IF ptrTc2_EtherCAT^.Input.Command.EcCoeSdoRead.Enable THEN
	FB_EcCoeSdoRead_0(
					sNetId		:= ptrTc2_EtherCAT^.Input.Parameter.EcCoeSdoRead.sNetId, 
					nSlaveAddr	:= ptrTc2_EtherCAT^.Input.Parameter.EcCoeSdoRead.nSlaveAddr, 
					nSubIndex	:= ptrTc2_EtherCAT^.Input.Parameter.EcCoeSdoRead.nSubIndex, 
					nIndex		:= ptrTc2_EtherCAT^.Input.Parameter.EcCoeSdoRead.nIndex , 
					pDstBuf		:= ptrTc2_EtherCAT^.Input.Parameter.EcCoeSdoRead.pDstBuf, 
					cbBufLen	:= ptrTc2_EtherCAT^.Input.Parameter.EcCoeSdoRead.cbBufLen, 
					bExecute	:= TRUE ,
					tTimeout	:= ptrTc2_EtherCAT^.Input.Parameter.EcCoeSdoRead.tTimeout, 
					bBusy		=> ptrTc2_EtherCAT^.Output.Status.EcCoeSdoRead.bBusy , 
					bError		=> ptrTc2_EtherCAT^.Output.Status.EcCoeSdoRead.bError, 
					nErrId		=> ptrTc2_EtherCAT^.Output.Error.ErrorID
					);
END_IF

IF NOT 	ptrTc2_EtherCAT^.Output.Status.EcCoeSdoRead.bBusy OR ptrTc2_EtherCAT^.Output.Status.EcCoeSdoRead.bError THEN
	ptrTc2_EtherCAT^.Input.Command.EcCoeSdoRead.Enable := FALSE ;
	FB_EcCoeSdoRead_0.bExecute := FALSE ;
	ptrTc2_EtherCAT^.Output.Status.EcCoeSdoRead.bError := FALSE ;
	FB_EcCoeSdoRead_0();
END_IF

(*IF ptrTc2_EtherCAT^.Input.Command.EcCoeSdoWrite.Enable THEN
	FB_EcCoESdoWrite_0(
						sNetId		:= ptrTc2_EtherCAT^.Input.Parameter.EcCoeSdoWrite.sNetId, 
						nSlaveAddr	:= ptrTc2_EtherCAT^.Input.Parameter.EcCoeSdoWrite.nSlaveAddr, 
						nSubIndex	:= ptrTc2_EtherCAT^.Input.Parameter.EcCoeSdoWrite.nSubIndex, 
						nIndex		:= ptrTc2_EtherCAT^.Input.Parameter.EcCoeSdoWrite.nIndex, 
						pSrcBuf		:= ptrTc2_EtherCAT^.Input.Parameter.EcCoeSdoWrite.pSrcBuf, 
						cbBufLen	:= ptrTc2_EtherCAT^.Input.Parameter.EcCoeSdoWrite.cbBufLen, 
						bExecute	:= TRUE, 
						tTimeout	:= ptrTc2_EtherCAT^.Input.Parameter.EcCoeSdoWrite.tTimeout, 
						bBusy		=> ptrTc2_EtherCAT^.Output.Status.EcCoeSdoWrite.bBusy, 
						bError		=> ptrTc2_EtherCAT^.Output.Status.EcCoeSdoWrite.bError, 
						nErrId		=> ptrTc2_EtherCAT^.Output.Error.ErrorID
					);			
END_IF

IF NOT 	ptrTc2_EtherCAT^.Output.Status.EcCoeSdoWrite.bBusy OR ptrTc2_EtherCAT^.Output.Status.EcCoeSdoWrite.bError THEN
	ptrTc2_EtherCAT^.Input.Command.EcCoeSdoWrite.Enable := FALSE ;
	FB_EcCoESdoWrite_0.bExecute := FALSE ;
	ptrTc2_EtherCAT^.Output.Status.EcCoeSdoWrite.bError := FALSE ;
	FB_EcCoESdoWrite_0();
END_IF	*)

IF ptrTc2_EtherCAT^.Input.Command.EcSoeRead.Enable THEN
	FB_EcSoERead_0(
					sNetId		:= ptrTc2_EtherCAT^.Input.Parameter.EcSoeRead.sNetId, 
					nSlaveAddr	:= ptrTc2_EtherCAT^.Input.Parameter.EcSoeRead.nSlaveAddr, 
					nIdn		:= ptrTc2_EtherCAT^.Input.Parameter.EcSoeRead.nIdn, 
					nElement	:= ptrTc2_EtherCAT^.Input.Parameter.EcSoeRead.nElement, 
					nDriveNo	:= ptrTc2_EtherCAT^.Input.Parameter.EcSoeRead.nDriveNo, 
					bCommand	:= ptrTc2_EtherCAT^.Input.Parameter.EcSoeRead.bCommand, 
					pDstBuf		:= ptrTc2_EtherCAT^.Input.Parameter.EcSoeRead.pDstBuf, 
					cbBufLen	:= ptrTc2_EtherCAT^.Input.Parameter.EcSoeRead.cbBufLen, 
					bExecute	:= ptrTc2_EtherCAT^.Input.Parameter.EcSoeRead.bExecute, 
					tTimeout	:= ptrTc2_EtherCAT^.Input.Parameter.EcSoeRead.tTimeout, 
					bBusy		=> ptrTc2_EtherCAT^.Output.Status.EcSoeRead.bBusy, 
					bError		=> ptrTc2_EtherCAT^.Output.Status.EcSoeRead.bError, 
					nErrId		=> ptrTc2_EtherCAT^.Output.Error.ErrorID 
				);
END_IF

IF ptrTc2_EtherCAT^.Input.Command.EcSoeWrite.Enable THEN
	FB_EcSoEWrite_0(
					sNetId		:= ptrTc2_EtherCAT^.Input.Parameter.EcSoeWrite.sNetId , 
					nSlaveAddr	:= ptrTc2_EtherCAT^.Input.Parameter.EcSoeWrite.nSlaveAddr, 
					nIdn		:= ptrTc2_EtherCAT^.Input.Parameter.EcSoeWrite.nIdn, 
					nElement	:= ptrTc2_EtherCAT^.Input.Parameter.EcSoeWrite.nElement, 
					nDriveNo	:= ptrTc2_EtherCAT^.Input.Parameter.EcSoeWrite.nDriveNo, 
					bCommand	:= ptrTc2_EtherCAT^.Input.Parameter.EcSoeWrite.pCommand, 
					pSrcBuf		:= ptrTc2_EtherCAT^.Input.Parameter.EcSoeWrite.pSrcBuf, 
					cbBufLen	:= ptrTc2_EtherCAT^.Input.Parameter.EcSoeWrite.cbBufLen, 
					bExecute	:= ptrTc2_EtherCAT^.Input.Parameter.EcSoeWrite.bExecute, 
					tTimeout	:= ptrTc2_EtherCAT^.Input.Parameter.EcSoeWrite.tTimeout, 
					bBusy		=> ptrTc2_EtherCAT^.Output.Status.EcSoeWrite.bBusy, 
					bError		=> ptrTc2_EtherCAT^.Output.Status.EcSoeWrite.bError, 
					nErrId		=> ptrTc2_EtherCAT^.Output.Error.ErrorID
				);
END_IF

METHOD EcCoeSdoWrite : BOOL
VAR_INPUT
END_VAR

VAR_INST
	bBusy:		BOOL;
END_VAR
IF ptrTc2_EtherCAT^.Input.Command.EcCoeSdoWrite.Enable THEN
	FB_EcCoeSdoWrite_0(
					sNetId		:= ptrTc2_EtherCAT^.Input.Parameter.EcCoeSdoWrite.sNetId, 
					nSlaveAddr	:= ptrTc2_EtherCAT^.Input.Parameter.EcCoeSdoWrite.nSlaveAddr, 
					nSubIndex	:= ptrTc2_EtherCAT^.Input.Parameter.EcCoeSdoWrite.nSubIndex, 
					nIndex		:= ptrTc2_EtherCAT^.Input.Parameter.EcCoeSdoWrite.nIndex, 
					pSrcBuf		:= ptrTc2_EtherCAT^.Input.Parameter.EcCoeSdoWrite.pSrcBuf, 
					cbBufLen	:= ptrTc2_EtherCAT^.Input.Parameter.EcCoeSdoWrite.cbBufLen, 
					bExecute	:= TRUE, 
					tTimeout	:= ptrTc2_EtherCAT^.Input.Parameter.EcCoeSdoWrite.tTimeout, 
					bBusy		=> ptrTc2_EtherCAT^.Output.Status.EcCoeSdoWrite.bBusy, 
					bError		=> ptrTc2_EtherCAT^.Output.Status.EcCoeSdoWrite.bError, 
					nErrId		=> ptrTc2_EtherCAT^.Output.Error.ErrorID
				);			

END_IF
				
IF ptrTc2_EtherCAT^.Output.Status.EcCoeSdoWrite.bBusy THEN
	bBusy:=	TRUE;
END_IF
	
IF bBusy AND NOT ptrTc2_EtherCAT^.Output.Status.EcCoeSdoWrite.bBusy  THEN
	bBusy:=		FALSE;
	ptrTc2_EtherCAT^.Input.Command.EcCoeSdoWrite.Enable:=	FALSE;
	FB_EcCoESdoWrite_0(bExecute := FALSE);
	IF (ptrTc2_EtherCAT^.Output.Status.EcCoeSdoWrite.bError = FALSE) THEN		
		EcCoeSdoWrite:= TRUE;
	END_IF
END_IF
END_METHOD

END_FUNCTION_BLOCK

// ---- POUs/Lib/Motion/External Libs/exARRAY_MAX.TcPOU
FUNCTION exARRAY_MAX : REAL
VAR_INPUT
	pt: POINTER TO ARRAY[0..32000] OF REAL;
	size: UINT;
END_VAR
VAR
	i: UINT;
	stop: UINT;
END_VAR

stop := (size -SIZEOF(pt)) / SIZEOF(pt);
exARRAY_MAX := pt^[0];
FOR i := 1 TO stop DO
	IF pt^[i] > exARRAY_MAX THEN exARRAY_MAX := pt^[i]; END_IF;
END_FOR;

(* revision history
hm	2. oct 2006		rev 1.0
	original version

hm	16. mar. 2008	rev 1.1
	changed input size to uint
*)

END_FUNCTION

// ---- POUs/Lib/Motion/External Libs/exARRAY_MIN.TcPOU
FUNCTION exARRAY_MIN : REAL
VAR_INPUT
	pt: POINTER TO ARRAY[0..32000] OF REAL;
	size: UINT;
END_VAR
VAR
	i: UINT;
	stop: UINT;
END_VAR

stop := (size - SIZEOF(pt)) / SIZEOF(pt);
exARRAY_MIN := pt^[0];
FOR i := 1 TO stop DO
	IF pt^[i] < exARRAY_MIN THEN exARRAY_MIN := pt^[i]; END_IF;
END_FOR;


(* revision history
hm		2. oct. 2006
	original version

hm		16. mar. 2008
	changed type of input size to uint

*)

END_FUNCTION

// ---- POUs/Lib/Motion/External Libs/exBIT_COUNT.TcPOU
FUNCTION exBIT_COUNT : INT
VAR_INPUT
	IN: DWORD;
END_VAR

WHILE in > 0 DO
	IF in.0 THEN exBit_Count := exBit_Count + 1; END_IF;
	in := SHR(in,1);
END_WHILE;



(* revision history
5.7.2007	rev 1.0		original version

10.9.2007	rev 1.1		hm
	changed algorithm for better performace
	the execution time has reduced by a factor of 5
	deleted unused variable temp
*)

END_FUNCTION

// ---- POUs/Lib/Motion/External Libs/exCHR_TO_STRING.TcPOU
FUNCTION exCHR_TO_STRING : STRING(1)
VAR_INPUT
	C: BYTE;
END_VAR
VAR
	PT: POINTER TO BYTE;
END_VAR

PT := ADR(exCHR_TO_STRING);
PT^ := C;
pt := pt + 1;
pt^ := 0;

(* revision history
hm	16 jan 2007		rev 1.0
	original version

hm	4. feb. 2008	rev 1.1
	return string would not be terminated properly

hm	29. mar. 2008	rev 1.2
	changed STRING to STRING(1)

hm	17. dec. 2008	rev 1.3
	changed name of function from chr to chr_to_string
*)

END_FUNCTION

// ---- POUs/Lib/Motion/External Libs/exDWORD_TO_STRF.TcPOU
FUNCTION exDWORD_TO_STRF : STRING(20)
VAR_INPUT
	IN: DWORD;
	N: INT;
END_VAR

(* limit N to max 20 characters *)
(* convert dword to string first and cut to length N *)
exDWORD_TO_STRF := exFIX(DWORD_TO_STRING(in),LIMIT(0,N,20),48,1);


(* revision history
hm	26. jan.2007	rev 1.0		
	original version

hm	29. mar. 2008	rev 1.1
	changed STRING to STRING(20)
	limit the output string to max 20 digits
*)

END_FUNCTION

// ---- POUs/Lib/Motion/External Libs/exFIX.TcPOU
FUNCTION exFIX : STRING(STRING_LENGTH)
VAR_INPUT
	str: STRING(STRING_LENGTH);
	L: INT;
	C: BYTE;
	M: INT;
END_VAR
VAR
	N: INT;
	SX: STRING(STRING_LENGTH);
END_VAR

(* make sure L does not exceed the limits of a string *)
N := LIMIT(0,L,STRING_LENGTH) - LEN(str);
IF N <= 0 THEN
	(* truncate the string at length N *)
	IF M = 1 THEN
		exFIX := RIGHT(str,L);
	ELSE
		exFIX := LEFT(str,L);
	END_IF;
ELSIF M = 1 THEN
	(* connect fill characters at the beginning *)
	sx := exFILL(C,N);
	exFIX := CONCAT(sx,str);
ELSIF M = 2 THEN
	(* center str beween fill characters *)
	(* for an uneven number of fill characters, there is one more at the end *)
	sx := exFILL(C,SHR(N+1,1));
	exFIX := CONCAT(str,sx);
	SX := LEFT(sx,SHR(N,1));
	exFIX := CONCAT(sx,exFIX);
ELSE
	(* connect fill characters at the end *)
	SX := exFILL(C,N);
	exFIX := CONCAT(str,SX);
END_IF;


(* revision histroy
hm	29. mar. 2008	rev 1.0
	original release

*)

END_FUNCTION

// ---- POUs/Lib/Motion/External Libs/exFILL.TcPOU
FUNCTION exFILL : STRING(STRING_LENGTH)
VAR_INPUT
	C: BYTE;
	L: INT;
END_VAR
VAR
	i: INT;
	sx: STRING(1);
END_VAR

Sx := exCHR_TO_STRING(c);
(* limit L to maximum 80 characters the length of a standard string *)
L := LIMIT(0,L,STRING_LENGTH);
(* create a string of characters to be connected to str *)
FOR i := 1 TO 8 DO
	exFILL := CONCAT(exFILL,exFILL);
	IF L.7 THEN exFILL := CONCAT(exFILL,Sx); END_IF;
	L := SHL(L,1);
END_FOR;




(* revision histroy
hm	29. mar. 2008	rev 1.0
	original release

hm	17. dec. 2008	rev 1.1
	changed function chr to chr_to_string

*)

END_FUNCTION

// ---- POUs/Lib/Motion/External Libs/exD_TRUNC.TcPOU
FUNCTION exD_TRUNC : DINT
VAR_INPUT
	X: REAL;
END_VAR

exD_TRUNC := REAL_TO_DINT(X);
IF X > 0.0 THEN
	IF DINT_TO_REAL(exD_TRUNC) > X THEN exD_TRUNC := exD_TRUNC - 1; END_IF;
ELSE
	IF DINT_TO_REAL(exD_TRUNC) < X THEN exD_TRUNC := exD_TRUNC + 1; END_IF;
END_IF;


(* for systems that support a dint truncation this routine can be replaced by trunc() *)


(* revision history
hm	21. mar. 2008	rev 1.0
	original version

hm	31. oct. 2008	rev 1.1
	optimized performance

hm	10. mar. 2009	rev 1.2
	real constants updated to new systax using dot
*)

END_FUNCTION

// ---- POUs/Lib/Motion/External Libs/exEVEN.TcPOU
FUNCTION exEVEN : BOOL
VAR_INPUT
	in: DINT;
END_VAR

exEVEN := NOT in.0;

(* revision history
hm	1. oct 2006	rev 1.0
	ORIGINAL VERSION

hm	01.12.2007	rev 1.1
	changed code for improved performance

hm	21. mar. 2008	rev 1.2
	changed type of input IN from INT to DINT
*)

END_FUNCTION

// ---- POUs/Lib/Motion/External Libs/exFRACT.TcPOU
FUNCTION exFRACT : REAL
VAR_INPUT
	x: REAL;
END_VAR

IF ABS(x) < 2.0E9 THEN
	exFRACT := x - DINT_TO_REAL(exD_TRUNC(x));
ELSE
	exFRACT := 0.0;
END_IF;

(* revision history
hm	4. aug 2006	rev 1.0
	original version

hm	11. mar 2008	rev 1.1
	added dint_to_real for compatibility reasons
	now returns 0 for number > 2e9
	changed input to x

hm	21. mar. 2008	rev 1.2
	use D_trunc instead of TRUNC for compatibility reasons

hm	10. mar. 2009	rev 1.3
	real constants updated to new systax using dot

*)

END_FUNCTION

// ---- POUs/Lib/Motion/External Libs/exF_POWER.TcPOU
FUNCTION exF_POWER : REAL
VAR_INPUT
	a: REAL;
	x: REAL;
	n: REAL;
END_VAR

exF_POWER := a * EXPT(X, N);

END_FUNCTION

// ---- POUs/Lib/Motion/External Libs/exINC1.TcPOU
FUNCTION exINC1 : INT
VAR_INPUT
	X: INT;
	N: INT;
END_VAR

IF X >= N - 1 THEN
	exINC1 := 0;
ELSE
	exINC1 := X + 1;
END_IF;



(* revision history
hm	13. oct. 2008	rev 1.0
	original version

hm	22. oct. 2008	rev 1.1
	added statement to return value for compatibility reasons

hm	23. feb. 2009	rev 1.2
 	when inc1 is called with X >= N inc will continue with 0
*)

END_FUNCTION

// ---- POUs/Lib/Motion/External Libs/exRDM.TcPOU
FUNCTION exRDM : REAL
VAR_INPUT
	last: REAL;
END_VAR
VAR
	tn: DWORD;
	tc: INT;
END_VAR

tn := exT_PLC_MS();
tc := exBIT_COUNT(tn);
tn.31 := tn.2;
tn.30 := tn.5;
tn.29 := tn.4;
tn.28 := tn.1;
tn.27 := tn.0;
tn.26 := tn.7;
tn.25 := tn.6;
tn.24 := tn.3;
tn := ROL(tn,exBIT_COUNT(tn)) OR 16#80000001;
tn := tn MOD 71474513 + INT_TO_DWORD(tc + 77);
exRDM := exFRACT(DWORD_TO_REAL(tn) / 10000000.0 * (math.E - LIMIT(0.0,last,1.0)));


(*
pt := ADR(temp);
pt^ := (T_PLC_MS() AND 16#007FFFFF) OR 16#3D000000;
RDM := fract(modR(temp*e+pi1, PI1-last) + modR(temp*PI1+e + last,e-last));
*)

(* revision history
hm		16. jan 2007		rev 1.0
	original version

hm		11. nov 2007		rev 1.1
	changed time() into t_plc_ms()

hm		20. nov 2007		rev 1.2
	changed code of temp calculation to avoid overflow in modr due to resuclt would not fit DINT for high timeer values

hm		5. jan 2008		rev 1.3
	changed calculation of temp to avoid problem with high values of t_plc_ms

hm		2. feb 2008		rev 1.4
	changed algorithm to avoind non iec functions and guarantee more randomness

hm	10. mar. 2008		rev 1.5
	make sure last will be between 0 and 1 to avoid invalid results

hm	16. mar. 2008		rev 1.6
	added conversion for tc to avoid warnings under codesys 3.0

hm	18. may. 2008		rev 1.7
	changed constant E to E1

hm	18. oct. 2008		rev 1.8
	using math constants

hm	10. mar. 2009		rev 1.9
	real constants updated to new systax using dot

*)

END_FUNCTION

// ---- POUs/Lib/Motion/External Libs/exT_PLC_MS.TcPOU
FUNCTION exT_PLC_MS : DWORD
VAR CONSTANT
	debug: BOOL := 0;
	N: INT := 0;
	offset: DWORD := 0;
END_VAR
VAR
	tx: TIME;
END_VAR

tx := TIME();
exT_PLC_MS := TIME_TO_DWORD(Tx);
(* hier muss die korrektur fr step7 stattfinden
plctime muss den vollen wertebereich von time ausnutzen:
wenn bei step7 time -24tage bis plus 24 tage ist dann muss der timer auch beim berlauf auf -24tage springen 
und auf keinen fall auf 0 !!!!
fr siemens muss ein weiterer fb im main eingebunden werden der sicherstellt das alle 32 bits durchgezהhlt werden.
es kann nur ein fb sein den er muss sich das oberste (32te) bit merken.
oder etwa spring s7 bei berlauf auf -24 tage????? dann wהre keine korrektur nצtig.
*)
IF debug THEN
	exT_PLC_MS := (SHL(exT_PLC_MS,N) OR SHL(DWORD#1,N)-1) + OFFSET;
END_IF;

(* revision history
hm	14.9.2007	rev 1.0
	original version

hm	12. nov 2007	rev 1.1
	added temporaray variable tx because some compilers could not handle time() as an argument

hm	16. nov. 2008	rev 1.2
	initialized constants with 0 for compatibility reasons
*)

END_FUNCTION

// ---- POUs/Lib/Motion/External Libs/exRDM2.TcPOU
FUNCTION exRDM2 : INT
VAR_INPUT
	last: INT;
	low: INT;
	high: INT;
END_VAR

exRDM2 := TRUNC_INT(exRDM(exFRACT(last * math.PI)) * (high - low + 1)) + low;

(* revision history
hm		29. feb 2008		rev 1.0
	original version

hm		18. oct. 2008		rev 1.1
	using math constants

*)

END_FUNCTION

// ---- POUs/Lib/Motion/External Libs/exTEMP_NTC.TcPOU
FUNCTION exTEMP_NTC : REAL
VAR_INPUT
	RES: REAL;	(* Resistance *)
	RN: REAL;	(* Thermistor Nominal -> Resistance At Room Temp -> 10K At 25c *)
	B: REAL;	(* Beta coeffiecent *)
END_VAR

IF res > 0.0 THEN
	exTEMP_NTC := B * 298.15 / (B + LN(RES / RN) * 298.15) -273.15;
END_IF;


(* revision history

hm 30. dec. 2008	rev 1.0
	original version

hm	11. mar. 2009	rev 1.1
	changed real constants to use dot syntax

*)

END_FUNCTION

// ---- POUs/Lib/Motion/External Libs/exTOGGLE.TcPOU
FUNCTION_BLOCK exTOGGLE
VAR_INPUT
	CLK: BOOL;
	rst: BOOL;
END_VAR
VAR_OUTPUT
	Q: BOOL;
END_VAR
VAR
	edge: BOOL;
END_VAR

IF rst THEN
	q := 0;
ELSIF clk AND NOT edge THEN
	Q := NOT Q;
END_IF;
edge := clk;

(* revision history

hm	13.9.2007		rev 1.0
	original version

hm	30. oct. 2008	rev 1.1
	deleted unnecessary init

*)

END_FUNCTION_BLOCK

// ---- POUs/Lib/Motion/External Libs/ex_ARRAY_MEDIAN.TcPOU
FUNCTION ex_ARRAY_MEDIAN : REAL
VAR_INPUT
	pt: POINTER TO ARRAY[0..32000] OF REAL;
	size: UINT;
END_VAR
VAR
	i: UINT;
	stop: UINT;
END_VAR

ex_ARRAY_SORT(pt,size);
stop := SHR(size,2)-1;
IF exEVEN(UINT_TO_INT(stop)) THEN
	ex_ARRAY_MEDIAN := pt^[SHR(stop,1)];
ELSE
	i := SHR(stop,1);
	ex_ARRAY_MEDIAN := (pt^[i] + pt^[i+1]) * 0.5;
END_IF;

(* old code
stop := (size - SIZEOF(pt)) / SIZEOF(pt);
FOR i := 0 TO stop - 1 DO
	FOR m := i + 1 TO stop DO
		IF pt^[i] > pt^[m] THEN
			temp := pt^[i];
			pt^[i] := pt^[m];
			pt^[m] := temp;
		END_IF;
	END_FOR;
END_FOR;
IF even(stop) THEN
	_array_median := pt^[stop/2];
ELSE
	i := stop/2;
	_array_median := (pt^[i] + pt^[i+1])/2;
END_IF;
*)
(* revision history
hm 	3.3.2007		rev 1.1
	corrected an error, changed the statement line 14	i := TRUNC(stop/2); to i := stop/2;

hm		22. sep 2007	rev 1.2
	changed algorithm to use _array_soft for performance reasons

hm		8. oct 2007		rev 1.3
	deleted unused variables m and temp

hm		14. nov 2007	rev 1.4
	corrected a problem with size calculation

hm		16.3. 2008		rev 1.5
	changed type of input size to uint
	performance improvements
*)

END_FUNCTION

// ---- POUs/Lib/Motion/External Libs/ex_ARRAY_SORT.TcPOU
FUNCTION ex_ARRAY_SORT : BOOL
VAR_INPUT
	PT: POINTER TO ARRAY[1..32000] OF REAL;
	SIZE: UINT;
END_VAR
VAR
	/// Laufvariable Stack
	stack_count: UINT;
	/// Stackgrצe~ 1,6*Log(n)/log(2) 
	stack: ARRAY[1..32] OF UINT;
	/// Anfangselement des Arrays 
	links: UINT;
	/// Endelement des Arrays 
	rechts: UINT;
	/// temporהrer Schwellwert fr Tauschbedingung 
	pivot: REAL;
	/// Laufvariable1 
	i: UINT;
	/// Laufvariable2 
	j: UINT;
	/// Ende innere Schleife 
	ende_innen: BOOL;
	/// Ende הuere Schleife 
	ende_aussen: BOOL;
	/// Hilfsvariable zum Tauschen von Werten 
	tmp: REAL;
END_VAR

(* Startwerte zur Arraygrצe *)
links := 1;					(* Anfangselement des Arrays *)
rechts := SHR(size,2);		(* Endelement des Arrays *)
stack_count := 1;			(* Laufvariable Stack *)

WHILE NOT ende_aussen DO						(* הuere Schleife *)
	IF links < rechts THEN
		pivot := PT^[SHR(rechts+links,1)];			(* Wert des mittleren Elements als Pivot-Wert *)
		i := links -1;
		j := rechts +1;

		(* innere Schleife, teile Feld *)
		ende_innen := FALSE;
		REPEAT

			(* steigende Reihenfolge *)
			REPEAT	i := i+1;	UNTIL (PT^[i] >= pivot) OR NOT (i < rechts)	END_REPEAT;
			REPEAT	j := j-1;	UNTIL (PT^[j] <= pivot) OR NOT (j > links)	END_REPEAT;


			(*sinkende Reihenfolge *)
(*			REPEAT	i := i+1;	UNTIL (PT^[i] <= pivot) OR NOT (i < rechts)	END_REPEAT	*)
(*			REPEAT	j := j-1;	UNTIL (PT^[j] >= pivot) OR NOT (j > links)	END_REPEAT	*)

			IF i >= j THEN
				ende_innen := TRUE;
			ELSE
				   tmp := PT^[j];
				PT^[j] := PT^[i];
				PT^[i] := tmp;
			END_IF;

		UNTIL ende_innen END_REPEAT;

		(* Push stack *)
		stack[stack_count] := rechts;		(* rechten Teil spהter sortieren *)
		IF Stack_count < 32 THEN
			stack_count := stack_count +1;
		ELSE
			ende_aussen := TRUE;
			ex_ARRAY_SORT := FALSE;					(* Fehler: Stack zu klein *)
		END_IF;

		(* linken Teil sortiern *)
		rechts := MAX(links, i-1);

	ELSE

		IF stack_count = 1 THEN
			ende_aussen := TRUE;
		ELSE

			links := rechts+1;

			(* pop stack *)
			stack_count := stack_count -1;		(* jetzt rechten Teil sortierne *)
			rechts:= stack[stack_count];
		END_IF;

	END_IF;

END_WHILE;

ex_ARRAY_SORT := TRUE;				(* Sortierung beendet *)


(* algorithm used before rev 2.0

size := SHR(size,2);
size2 := UINT_TO_INT(SHR(size,1));
FOR i := SIZE2  TO 1 BY -1 DO
	j:=i;
    WHILE j <= SIZE2 DO
     	stop := j * 2 + 1;
        IF stop > UINT_TO_INT(SIZE) THEN stop := stop - 1;
        ELSIF pt^[stop-1] > pt^[stop] THEN stop := stop - 1;
		END_IF;
        IF pt^[j] < pt^[stop] THEN
         	temp := pt^[j];
            pt^[j] := pt^[stop];
            pt^[stop] := temp;
        END_IF;
        j := stop;
    END_WHILE;
END_FOR;

*)

(* heapsort
FOR heapsize := UINT_TO_INT(size) TO 1 BY -1 DO
	popmax := pt^[1];
	pt^[1] := pt^[heapsize];
   	i := 1;
	hs2 := SHR(heapsize,1);
	WHILE i <= hs2 DO
       	stop := i * 2 + 1;  
        	IF stop > heapsize THEN stop := stop - 1;
        	ELSIF pt^[stop-1] > pt^[stop] THEN stop := stop - 1;
	 	END_IF;
        	IF pt^[i] < pt^[stop] THEN
            		temp := pt^[i];
            		pt^[i] := pt^[stop];
            		pt^[stop] := temp;
        	END_IF;
        	i := stop;
    	END_WHILE;
	pt^[heapsize] := popmax;
END_FOR;

_ARRAY_SORT2 := TRUE;
*)

(* old algorithm bubble sort used before rev 1.2
stop := (size - SIZEOF(pt)) / SIZEOF(pt);
FOR i := 0 TO stop - 1 DO
	FOR m := i + 1 TO stop DO
		IF pt^[i] > pt^[m] THEN
			temp := pt^[i];
			pt^[i] := pt^[m];
			pt^[m] := temp;
		END_IF;
	END_FOR;
END_FOR;
_array_sort := TRUE;

*)


(* revision history

hm 	6.1.2007 	rev 1.1
	changed return value to true

hm	22. sep 2007	rev 1.2
	changed sorting algorithm to heap sort for performance reasons

hm 	14. nov 2007	rev 1.3
	changed calculation of stop to be more efficient

hm	15 dec 2007	rev 1.4
	added function return true

hm	5. jan 2008		rev 1.5
	improved performance

hm	16. mar. 2008	rev 1.6
	changed type of input size to uint

hm	28. mar. 2008	rev 1.7
	changed input f to pt

hm	19. jan. 2011	rev 2.0
	new faster algorithm using qucksort (Alexander Drikitis)

*)

END_FUNCTION

// ---- POUs/Lib/Motion/External Libs/ex_ARRAY_SORT_LREAL.TcPOU
FUNCTION ex_ARRAY_SORT_LREAL : BOOL
VAR_INPUT
	PT: POINTER TO ARRAY[1..32000] OF LREAL;
	SIZE: UINT;
END_VAR
VAR
	/// Laufvariable Stack
	stack_count: UINT;
	/// Stackgrצe~ 1,6*Log(n)/log(2) 
	stack: ARRAY[1..256] OF UINT;
	/// Anfangselement des Arrays 
	links: UINT;
	/// Endelement des Arrays 
	rechts: UINT;
	/// temporהrer Schwellwert fr Tauschbedingung 
	pivot: LREAL;
	/// Laufvariable1 
	i: UINT;
	/// Laufvariable2 
	j: UINT;
	/// Ende innere Schleife 
	ende_innen: BOOL;
	/// Ende הuere Schleife 
	ende_aussen: BOOL;
	/// Hilfsvariable zum Tauschen von Werten 
	tmp: LREAL;
END_VAR

(* Startwerte zur Arraygrצe *)
links := 1;					(* Anfangselement des Arrays *)
rechts := SHR(size,3);		(* Endelement des Arrays *)
stack_count := 1;			(* Laufvariable Stack *)

WHILE NOT ende_aussen DO						(* הuere Schleife *)
	IF links < rechts THEN
		pivot := PT^[SHR(rechts+links,1)];			(* Wert des mittleren Elements als Pivot-Wert *)
		i := links -1;
		j := rechts +1;

		(* innere Schleife, teile Feld *)
		ende_innen := FALSE;
		REPEAT

			(* steigende Reihenfolge *)
			REPEAT	i := i+1;	UNTIL (PT^[i] >= pivot) OR NOT (i < rechts)	END_REPEAT;
			REPEAT	j := j-1;	UNTIL (PT^[j] <= pivot) OR NOT (j > links)	END_REPEAT;


			(*sinkende Reihenfolge *)
(*			REPEAT	i := i+1;	UNTIL (PT^[i] <= pivot) OR NOT (i < rechts)	END_REPEAT	*)
(*			REPEAT	j := j-1;	UNTIL (PT^[j] >= pivot) OR NOT (j > links)	END_REPEAT	*)

			IF i >= j THEN
				ende_innen := TRUE;
			ELSE
				   tmp := PT^[j];
				PT^[j] := PT^[i];
				PT^[i] := tmp;
			END_IF;

		UNTIL ende_innen END_REPEAT;

		(* Push stack *)
		stack[stack_count] := rechts;		(* rechten Teil spהter sortieren *)
		IF Stack_count < 32 THEN
			stack_count := stack_count +1;
		ELSE
			ende_aussen := TRUE;
			ex_ARRAY_SORT_LREAL := FALSE;					(* Fehler: Stack zu klein *)
		END_IF;

		(* linken Teil sortiern *)
		rechts := MAX(links, i-1);

	ELSE

		IF stack_count = 1 THEN
			ende_aussen := TRUE;
		ELSE

			links := rechts+1;

			(* pop stack *)
			stack_count := stack_count -1;		(* jetzt rechten Teil sortierne *)
			rechts:= stack[stack_count];
		END_IF;

	END_IF;

END_WHILE;

ex_ARRAY_SORT_LREAL := TRUE;				(* Sortierung beendet *)


(* algorithm used before rev 2.0

size := SHR(size,2);
size2 := UINT_TO_INT(SHR(size,1));
FOR i := SIZE2  TO 1 BY -1 DO
	j:=i;
    WHILE j <= SIZE2 DO
     	stop := j * 2 + 1;
        IF stop > UINT_TO_INT(SIZE) THEN stop := stop - 1;
        ELSIF pt^[stop-1] > pt^[stop] THEN stop := stop - 1;
		END_IF;
        IF pt^[j] < pt^[stop] THEN
         	temp := pt^[j];
            pt^[j] := pt^[stop];
            pt^[stop] := temp;
        END_IF;
        j := stop;
    END_WHILE;
END_FOR;

*)

(* heapsort
FOR heapsize := UINT_TO_INT(size) TO 1 BY -1 DO
	popmax := pt^[1];
	pt^[1] := pt^[heapsize];
   	i := 1;
	hs2 := SHR(heapsize,1);
	WHILE i <= hs2 DO
       	stop := i * 2 + 1;  
        	IF stop > heapsize THEN stop := stop - 1;
        	ELSIF pt^[stop-1] > pt^[stop] THEN stop := stop - 1;
	 	END_IF;
        	IF pt^[i] < pt^[stop] THEN
            		temp := pt^[i];
            		pt^[i] := pt^[stop];
            		pt^[stop] := temp;
        	END_IF;
        	i := stop;
    	END_WHILE;
	pt^[heapsize] := popmax;
END_FOR;

_ARRAY_SORT2 := TRUE;
*)

(* old algorithm bubble sort used before rev 1.2
stop := (size - SIZEOF(pt)) / SIZEOF(pt);
FOR i := 0 TO stop - 1 DO
	FOR m := i + 1 TO stop DO
		IF pt^[i] > pt^[m] THEN
			temp := pt^[i];
			pt^[i] := pt^[m];
			pt^[m] := temp;
		END_IF;
	END_FOR;
END_FOR;
_array_sort := TRUE;

*)


(* revision history

hm 	6.1.2007 	rev 1.1
	changed return value to true

hm	22. sep 2007	rev 1.2
	changed sorting algorithm to heap sort for performance reasons

hm 	14. nov 2007	rev 1.3
	changed calculation of stop to be more efficient

hm	15 dec 2007	rev 1.4
	added function return true

hm	5. jan 2008		rev 1.5
	improved performance

hm	16. mar. 2008	rev 1.6
	changed type of input size to uint

hm	28. mar. 2008	rev 1.7
	changed input f to pt

hm	19. jan. 2011	rev 2.0
	new faster algorithm using qucksort (Alexander Drikitis)

*)

END_FUNCTION

// ---- POUs/Lib/Motion/External Libs/ex_ARRAY_SUM.TcPOU
FUNCTION ex_ARRAY_SUM : REAL
VAR_INPUT
	pt: POINTER TO ARRAY[0..32000] OF REAL;
	size: UINT;
END_VAR
VAR
	i: UINT;
	stop: UINT;
END_VAR

stop := (size -SIZEOF(pt)) / SIZEOF(pt);
ex_ARRAY_SUM := pt^[0];
FOR i := 1 TO stop DO
	ex_ARRAY_SUM := ex_ARRAY_SUM + pt^[i];
END_FOR;

(* revision history
hm 	2. oct. 2006	rev 1.0
	function created

hm	16. mar. 2008	rev 1.1
	changed type of input size to uint

*)

END_FUNCTION

// ---- POUs/Lib/Motion/FailureRport/Terminal/Group/TerminalGroupReport_FB.TcPOU
FUNCTION_BLOCK TerminalGroupReport_FB
VAR_INPUT
	Enable 				: BOOL;
	pGroupCtrl			: POINTER TO Terminal_Group_Ctrl_typ ;
	Ref_ev_Module_Event : REFERENCE TO ev_MOTOR_POSITION_ERROR REF= ev_MOTOR_POSITION_ERROR;
END_VAR
VAR_IN_OUT
	In 		: ARRAY[*]OF Terminal_Ctrl_typ ;	
	//Out		: ARRAY[*]OF ErrCollector_Out ;
END_VAR

VAR
	LogMsgInit          : BOOL := TRUE;
	LogMsg_0 			: LogMsg ;
	//Get old events from Q
	ExecuteTrig: 		Trigger;	
	WrongState :   		BOOL;
	nI         : DINT;
	InFault    : BOOL;
	
	fbPrgmBasic :FB_PrgmBasic;
	
	
	//Debug
	intErrorCounter : USINT := 0;
	
	LowerBound         : DINT;
END_VAR






IF pGroupCtrl <> 0 THEN
		
	IF LogMsgInit THEN      
		LogMsgInit := FALSE ;
		fnLogMsgInit(ADR(LogMsg_0), pGroupCtrl^.In.Par.GroupName, ADR(LogGlobalArray), ADR(CONST_ZERO));
		LogMsg_0.Enable:= 		TRUE;
	END_IF

	IF Enable THEN
		InFault := FALSE;
		
		LowerBound := LOWER_BOUND(In,1);
		
		FOR nI:= LOWER_BOUND(In,1) TO UPPER_BOUND(In,1) DO

	
			IF 	In[nI].In.Par.Name <> 'Empty' THEN
							
				// IF already in error reset others status
				IF InFault THEN
					In[nI].Out.Status.Fault := FALSE;
				ELSE	
					//If terminal is not on OPER state
					IF ((In[nI].Out.Status.TerminalState AND eTerminalStates.OP) = 0) THEN
							
						IF In[nI].Out.Status.Active THEN
							InFault := TRUE;												
							
							IF In[nI].Out.Status.Fault = FALSE THEN
								Meth_SetError(nI);							
							END_IF
						ELSE // Module Not Active
							
							Meth_HandleModuleNotActive(nI);										
						END_IF
						In[nI].Out.Status.Fault := TRUE;
					ELSE
						In[nI].Out.Status.Fault := FALSE;		
					END_IF
				
						
				END_IF
				In[nI].Out.Status.Active := 0;
				In[nI].Out.Monitor.SubSysName := '';
			END_IF
			
		END_FOR
		
		IF NOT InFault THEN
			pGroupCtrl^.Out.Status.errorBit := 0;
		END_IF	
		
		// Reset if for was brake	
		In[nI].Out.Status.Active := 0;
		In[nI].Out.Monitor.SubSysName := '';
	END_IF
	
	

END_IF	
fbPrgmBasic();
//fnLogTransfer FUNCTION call
fnLogTransfer(ADR(LogMsg_0));

METHOD Meth_HandleModuleNotActive : BOOL
VAR_INPUT
	
	NonActiveIndex: DINT;
	
END_VAR
VAR
	internalIndex : DINT;
END_VAR
	//if last
	IF NonActiveIndex = UPPER_BOUND(In,1) THEN
		//	System is OK because it is last
					
		//If next is not OK
	ELSIF In[nI+1].Out.Status.TerminalState <> eTerminalStates.OP THEN
		IF In[nI+1].Out.Status.Active THEN
			InFault := TRUE;	
			//next is Active and not OK
			IF In[NonActiveIndex].Out.Status.Fault = FALSE THEN
				Meth_SetError(NonActiveIndex);											
			END_IF											
			InFault := TRUE;
		ELSE// Check if there is active module after the problematic module
			FOR internalIndex:= NonActiveIndex TO UPPER_BOUND(In,1) DO
				IF In[internalIndex].Out.Status.Active THEN
					InFault := TRUE;	
					IF In[NonActiveIndex].Out.Status.Fault = FALSE THEN
						Meth_SetError(NonActiveIndex);											
					END_IF	
				END_IF		
			END_FOR
		END_IF
		
									
	ELSE 
			//Continue the next module is OK	;
		 	
	END_IF
END_METHOD

METHOD Meth_SendEvent : BOOL
VAR_INPUT
	RefEvent : REFERENCE TO EventHelper;
END_VAR
VAR
	EventParameters:EventParam_Typ;	
	EventHeader:EventHeader_Typ;	
	Dummy :DINT :=0;
//	pFlowID :POINTER TO DINT;
END_VAR
IF __ISVALIDREF(RefEvent) THEN
		
		EventHeader.SubsysID :=		pGroupCtrl^.In.Par.GroupID  ; 
 
		EventParameters.MotorID := 		 In[nI].In.Par.ModuleID; 	// Motor ID

		fbPrgmBasic.mEventThrow(RefEvent,ADR(EventHeader),ADR(EventParameters) );			//RefEvent();
		Meth_SendEvent := TRUE;
		
		


		//Debug
		intErrorCounter := intErrorCounter + 1;
		
END_IF
END_METHOD

METHOD Meth_SetError : BOOL
VAR_INPUT
	
	TerminalIndex: DINT;
	
END_VAR
VAR
	BitBase : ULINT ;
END_VAR
Meth_SendEvent(Ref_ev_Module_Event);

fnLogMsg(ADR(LogMsg_0), LOG_INFO, 'Terminal Error Q Send Group ID %d,In[nI].In.Par.ModuleID =%d',
							pGroupCtrl^.In.Par.GroupID  ,
							In[TerminalIndex].In.Par.ModuleID,							
							0);

							
BitBase := 2;			
pGroupCtrl^.Out.Status.errorBit := SHL(BitBase,(TerminalIndex -LowerBound));
END_METHOD

END_FUNCTION_BLOCK

// ---- POUs/Lib/Motion/ParIDAccess_FB.TcPOU
FUNCTION_BLOCK PUBLIC ParIDAccess_FB
VAR_INPUT
	
	BasicAxisCtrlPtr 	: POINTER TO Basic_axis_typ ;
	ParIDAccessCtrlPtr 	: POINTER TO ParIDAccess_Typ ;
	
END_VAR
VAR_IN_OUT

END_VAR
VAR_OUTPUT
END_VAR
	
VAR
	LogMsgInit		: BOOL := TRUE;
	LogMsg_0 		: LogMsg ;	
	
	fbGetCurTaskIdx: 		GETCURTASKINDEX;
    TaskCycleTimeUDINT: 	UDINT;
    TaskCycleTime: 			TIME;
	
	DisableTriger	: Trigger ;

	FB_EcCoeSdoRead_0 	: FB_EcCoeSdoRead;
	FB_EcCoeSdoWrite_0 	: FB_EcCoeSdoWrite;
	StateCoeSdoRead		: UINT;
	StateCoeSdoWrite	: UINT;	
	
	ErrorTrig : Trigger ;
	AxisStep : eParIDAccessState ;
	tempTrig : Trigger ;
			
	tmp_ErrorEntry			: Eh_ErrorEntry_typ;
	
END_VAR

IF LogMsgInit THEN 
	LogMsg_0.ptrGlobalArray		:= 	ADR(LogGlobalArray);
	LogMsg_0.ptrEncoderAngle	:= 	ADR(BasicAxisCtrlPtr^.Input.Parameter.PosForLog);   
	LogMsg_0.Enable:= 	TRUE; 	
	LogMsgInit	:= FALSE;
END_IF
LogMsg_0.logData.category	:=	BasicAxisCtrlPtr^.Input.Parameter.ThreadName;  

IF (TaskCycleTimeUDINT = 0) THEN
	fbGetCurTaskIdx();
	TaskCycleTimeUDINT := _TaskInfo[fbGetCurTaskIdx.index].CycleTime;
	TaskCycleTime	:= UDINT_TO_TIME(TaskCycleTimeUDINT/10000); 
END_IF 

IF BasicAxisCtrlPtr^.Output.Status.FAULT THEN
	
	THIS^.ResetAll_MC_FB();

	AxisStep := ParID_STATE_ERROR;
		
END_IF


CASE AxisStep OF
		
	(******************** WAIT *************************)
	ParID_STATE_WAIT:  (* STATE: Wait *)
		
		IF BasicAxisCtrlPtr^.Output.Status.ReadyForCmd THEN
			AxisStep := ParID_STATE_READY;
		END_IF
		
		THIS^.ResetAll_MC_FB();

	(******************** READY *************************)
	ParID_STATE_READY:
		
		IF (ParIDAccessCtrlPtr^.Input.Command.ReadCoeSdo = TRUE) THEN
			THIS^.EcCoeSdoRead(FALSE);
			AxisStep := ParID_STATE_READ_SDO; 
			
		ELSIF (ParIDAccessCtrlPtr^.Input.Command.WriteCoeSdo = TRUE) THEN
			THIS^.EcCoeSdoWrite(FALSE);
			AxisStep := ParID_STATE_WRITE_SDO; 
			

		END_IF
	
	(******************** Read Sdo **********************)
	ParID_STATE_READ_SDO:
	
		IF THIS^.EcCoeSdoRead(TRUE) THEN
			AxisStep := ParID_STATE_READY;
		END_IF
		
	(******************** Write Sdo **********************)
		
	ParID_STATE_WRITE_SDO:
	
		IF THIS^.EcCoeSdoWrite(TRUE) THEN
			AxisStep := ParID_STATE_READY;
		END_IF
		
		
	(******************** Error **********************)	
	ParID_STATE_ERROR:	
	
		THIS^.ResetAll_MC_FB();	
		
		IF BasicAxisCtrlPtr^.Output.Status.FAULT THEN
					
			AxisStep := ParID_STATE_ERROR;
		ELSE
			ParIDAccessCtrlPtr^.Output.Error.ErrorID := 0 ;
			AxisStep := ParID_STATE_WAIT;
		END_IF
	
	
END_CASE 
	
//=====================================================================================================================\\


//fnLogTransfer FUNCTION call
fnLogTransfer(ADR(LogMsg_0));

METHOD AddNCError : BOOL
VAR_INPUT
	ErrorId			: UDINT;
	ErrorPrefix     : STRING[100];
END_VAR

	tmp_ErrorEntry.ErrorId		:= ErrorId;

	tmp_ErrorEntry.ErrorText	:= ErrorPrefix;

	tmp_ErrorEntry.ErrorText	:= CONCAT(tmp_ErrorEntry.ErrorText, UDINT_TO_STRING(tmp_ErrorEntry.ErrorId));
	tmp_ErrorEntry.ErrorText	:= CONCAT(tmp_ErrorEntry.ErrorText, 'Task: ');
	tmp_ErrorEntry.ErrorText	:= CONCAT(tmp_ErrorEntry.ErrorText, ParIDAccessCtrlPtr^.Input.Parameter.ThreadName);	
	tmp_ErrorEntry.ErrorText	:= CONCAT(tmp_ErrorEntry.ErrorText, FC_NcErrorMsg(tmp_ErrorEntry.ErrorId));	
	fnLogMsg(ADR(LogMsg_0),LOG_ERROR,tmp_ErrorEntry.ErrorText,0,0,0);	
	
	tmp_ErrorEntry.MotorEvents := CreateNCErrMsgDetails(tmp_ErrorEntry.ErrorId);
	
	BasicAxisCtrlPtr^.Output.Error.fbErrorHandler.ErrorPush(tmp_ErrorEntry);
END_METHOD

METHOD EcCoeSdoRead : BOOL
VAR_INPUT
	Execute: 	BOOL;
END_VAR

VAR_INST
	errorTrig: 		Trigger ;	
	ExecuteTrig: 	Trigger;
END_VAR

IF ExecuteTrig.EDGEPOS(Execute) THEN
	ParIDAccessCtrlPtr^.Input.Command.ReadCoeSdo 	:= FALSE;
	EcCoeSdoRead:= FALSE;
	StateCoeSdoRead	:= 1;		
END_IF

IF ExecuteTrig.EDGENEG(Execute) THEN
	
	ParIDAccessCtrlPtr^.Output.Status.ReadCoeSdo.Done 	:= FALSE;
	FB_EcCoeSdoRead_0.bExecute 							:= FALSE;
	StateCoeSdoRead		:= 0;	
	EcCoeSdoRead		:= FALSE;
	
END_IF


CASE StateCoeSdoRead OF
	
	0:
		// Wait	
	1:
	
		FB_EcCoeSdoRead_0.sNetId		:= F_CreateAmsNetId(BasicAxisCtrlPtr^.Input.Parameter.ecNetIdArr); 
		FB_EcCoeSdoRead_0.nSlaveAddr	:= LREAL_TO_UINT(BasicAxisCtrlPtr^.Input.Parameter.Drive.EtherCatAddr);
		FB_EcCoeSdoRead_0.nSubIndex		:= ParIDAccessCtrlPtr^.Input.Parameter.ReadCoedSdo.nSubIndex;
		FB_EcCoeSdoRead_0.nIndex		:= ParIDAccessCtrlPtr^.Input.Parameter.ReadCoedSdo.nIndex; 
		FB_EcCoeSdoRead_0.pDstBuf		:= ParIDAccessCtrlPtr^.Input.Parameter.ReadCoedSdo.pDstBuf; 
		FB_EcCoeSdoRead_0.cbBufLen		:= ParIDAccessCtrlPtr^.Input.Parameter.ReadCoedSdo.cbBufLen; 
		FB_EcCoeSdoRead_0.tTimeout		:= ParIDAccessCtrlPtr^.Input.Parameter.ReadCoedSdo.tTimeout; 
		StateCoeSdoRead	:= 2;	
	2:	

		FB_EcCoeSdoRead_0.bExecute		:= TRUE;	
		IF (FB_EcCoeSdoRead_0.bBusy = TRUE) THEN
			StateCoeSdoRead	:= 3;	
		END_IF

	3:	
		IF (FB_EcCoeSdoRead_0.bBusy = FALSE) THEN
			FB_EcCoeSdoRead_0.bExecute		:= FALSE;
			ParIDAccessCtrlPtr^.Output.Status.ReadCoeSdo.Done	:= TRUE;
			EcCoeSdoRead	:= TRUE;
			StateCoeSdoRead	:= 0;	
		END_IF
	
END_CASE

FB_EcCoeSdoRead_0();

(* check if error occured *)
IF errorTrig.EDGEPOS(FB_EcCoeSdoRead_0.bError) THEN
	
	// Add FB Error to ErrorHandler	
	AddNCError(FB_EcCoeSdoRead_0.nErrId,'NC Error FB_EcCoeSdoRead_0 ErrorID: ');
	
	EcCoeSdoRead :=  FALSE ;
	ParIDAccessCtrlPtr^.Input.Command.ReadCoeSdo := FALSE;
	FB_EcCoeSdoRead_0.bExecute := FALSE;
END_IF

ParIDAccessCtrlPtr^.Output.Status.ReadCoeSdo.Busy	:= FB_EcCoeSdoRead_0.bBusy;
END_METHOD

METHOD EcCoeSdoWrite : BOOL
VAR_INPUT
	Execute: 	BOOL;
END_VAR

VAR_INST
	errorTrig: 		Trigger ;	
	ExecuteTrig: 	Trigger;
END_VAR

IF ExecuteTrig.EDGEPOS(Execute) THEN
	ParIDAccessCtrlPtr^.Input.Command.WriteCoeSdo 		:= FALSE;
	EcCoeSdoWrite		:= FALSE;
	StateCoeSdoWrite	:= 1;		
END_IF

IF ExecuteTrig.EDGENEG(Execute) THEN
	
	ParIDAccessCtrlPtr^.Output.Status.WriteCoeSdo.Done := FALSE;
	FB_EcCoeSdoWrite_0.bExecute 				:= FALSE;
	StateCoeSdoWrite	:= 0;	
	EcCoeSdoWrite		:= FALSE;
	
END_IF


CASE StateCoeSdoWrite OF
	
	0:
		// Wait	
	1:
	
		FB_EcCoeSdoWrite_0.sNetId		:= F_CreateAmsNetId(BasicAxisCtrlPtr^.Input.Parameter.ecNetIdArr); 
		FB_EcCoeSdoWrite_0.nSlaveAddr	:= BasicAxisCtrlPtr^.Input.Parameter.Drive.EtherCatAddr;
		FB_EcCoeSdoWrite_0.nSubIndex	:= ParIDAccessCtrlPtr^.Input.Parameter.WriteCoeSdo.nSubIndex;
		FB_EcCoeSdoWrite_0.nIndex		:= ParIDAccessCtrlPtr^.Input.Parameter.WriteCoeSdo.nIndex; 
		FB_EcCoeSdoWrite_0.pSrcBuf		:= ParIDAccessCtrlPtr^.Input.Parameter.WriteCoeSdo.pSrcBuf; 
		FB_EcCoeSdoWrite_0.cbBufLen		:= ParIDAccessCtrlPtr^.Input.Parameter.WriteCoeSdo.cbBufLen; 
		FB_EcCoeSdoWrite_0.tTimeout		:= ParIDAccessCtrlPtr^.Input.Parameter.WriteCoeSdo.tTimeout; 
		StateCoeSdoWrite	:= 2;	
	2:	

		FB_EcCoeSdoWrite_0.bExecute		:= TRUE;	
		IF (FB_EcCoeSdoWrite_0.bBusy = TRUE) THEN
			StateCoeSdoWrite	:= 3;	
		END_IF

	3:	
		IF (FB_EcCoeSdoWrite_0.bBusy = FALSE) THEN
			FB_EcCoeSdoWrite_0.bExecute		:= FALSE;
			ParIDAccessCtrlPtr^.Output.Status.WriteCoeSdo.Done	:= TRUE;
			EcCoeSdoWrite		:= TRUE;
			StateCoeSdoWrite	:= 0;	
		END_IF
	
END_CASE

FB_EcCoeSdoWrite_0();

(* check if error occured *)
IF errorTrig.EDGEPOS(FB_EcCoeSdoWrite_0.bError) THEN
	
	// Add FB Error to ErrorHandler	
	AddNCError(FB_EcCoeSdoWrite_0.nErrId,'NC Error FB_EcCoeSdoWrite_0 ErrorID: ');
	
	EcCoeSdoWrite :=  FALSE ;
	ParIDAccessCtrlPtr^.Input.Command.WriteCoeSdo := FALSE;
	FB_EcCoeSdoWrite_0.bExecute := FALSE;
END_IF

ParIDAccessCtrlPtr^.Output.Status.WriteCoeSdo.Busy	:= FB_EcCoeSdoWrite_0.bBusy;
END_METHOD

METHOD PRIVATE ResetAll_MC_FB : BOOL
VAR_INPUT
END_VAR

		ResetAll_MC_FB := FALSE ;
				
		FB_EcCoeSdoRead_0.bExecute	:= FALSE;
		FB_EcCoeSdoWrite_0.bExecute	:= FALSE;
		{warning disable C0371}
		//Warning: Access to VAR_IN_OUT <Var> declared in <POU> from external context <Method/Transition/Property>
		FB_EcCoeSdoRead_0(); 
		FB_EcCoeSdoWrite_0() ;
		{warning restore C0371}
		
		
		memset(ADR(ParIDAccessCtrlPtr^.Input.Command) ,0 ,SIZEOF(ParIDAccessCtrlPtr^.Input.Command));
		memset(ADR(ParIDAccessCtrlPtr^.Output.Status) ,0 ,SIZEOF(ParIDAccessCtrlPtr^.Output.Status));
		
		ResetAll_MC_FB := TRUE ;
END_METHOD

END_FUNCTION_BLOCK

// ---- POUs/Lib/Signal/FB_LPF.TcPOU
FUNCTION_BLOCK FB_LPF
VAR_INPUT
	IN:	LREAL;	// Input
	Fc:	LREAL;	// Frequecy
END_VAR
VAR_OUTPUT
	OUT:	LREAL;
END_VAR
VAR
	
 	fbGetCurTaskIdx: 		GETCURTASKINDEX;
 	TaskCycleTimeUDINT: 	UDINT;
	DeltaT:	LREAL;
	RC:		LREAL;
	A:		LREAL;
END_VAR

VAR CONSTANT	 	 		
	
	PI:	REAL:=3.14159265;
	
END_VAR

// Xi - Current input value
// Yi-1 - Last Result
//Yi - New Result
// Yi = A*Xi + (1-A)*Yi-1

IF (TaskCycleTimeUDINT = 0) THEN
	fbGetCurTaskIdx();
	TaskCycleTimeUDINT := _TaskInfo[fbGetCurTaskIdx.index].CycleTime;
	DeltaT	:= UDINT_TO_LREAL(TaskCycleTimeUDINT)/10000000; 
END_IF

RC	:= 1/(2*PI*Fc);
A	:= DeltaT/(RC + DeltaT);

OUT	:= A*IN + (1-A)*OUT;

END_FUNCTION_BLOCK

// ---- POUs/Lib/System/CmdQueue/FB_CmdQueue.TcPOU

(*
	Add command by order, queue will scan only the head, this can be changed in the future.
	Element type type should be with a struct which contains DelayInfo_typ at start.  
*)

FUNCTION_BLOCK FB_CmdQueue
VAR_INPUT
	
	pBufferPool		: PVOID;
	BufferSize		: UDINT;
	ElementSize		: UDINT;
	rLogMsg 		: REFERENCE TO LogMsg ;
	Name : STRING := 'CmdQueue';			
	Position	:ULINT;
END_VAR
VAR_OUTPUT
END_VAR
VAR

	InitDone : BOOL;
	NumElements : UDINT;
	
	HeadIndex : UDINT; // index from 0
	TailIndex : UDINT; // index from 0
	UsedSize  : UDINT;
		
	MutexFlag : BOOL;
	
END_VAR

VAR_STAT
END_VAR

IF NOT InitDone THEN
	mInit();
	InitDone := TRUE;
END_IF

METHOD PUBLIC mAdd : BOOL
VAR_INPUT
	pElement		: PVOID;
END_VAR

VAR
	NewElementIndex : UDINT;
	
	pDelayedCmdInfo : POINTER TO DelayInfo_typ;
END_VAR

VAR_STAT
    sRid : UDINT := 1111;
END_VAR

IF NOT TestAndSet(MutexFlag) THEN
	RETURN;
END_IF

IF mIsFull() THEN
	MutexFlag := FALSE;
	RETURN;
END_IF

IF mIsEmpty() THEN
	NewElementIndex := TailIndex;	
ELSE
	NewElementIndex := (TailIndex + 1) MOD NumElements;
END_IF

TailIndex := NewElementIndex;
UsedSize := UsedSize + 1;

pDelayedCmdInfo := pElement;
pDelayedCmdInfo^.GroupId := pDelayedCmdInfo^.RequestId := sRid;
sRid := sRid+1;

IF (pDelayedCmdInfo^.pExecuted <> 0) THEN
//	pDelayedCmdInfo^.pExecuted^ := FALSE;
END_IF

pDelayedCmdInfo^.Executed := FALSE;
pDelayedCmdInfo^.LagError := 0;

MEMCPY((pBufferPool + NewElementIndex * ElementSize), pElement, ElementSize);

MutexFlag := FALSE;

mAdd := TRUE;
END_METHOD

METHOD PUBLIC mCheck : PVOID // will return true only when next cmd will be ready (time/pos is up)
VAR_INPUT
END_VAR

IF NOT TestAndSet(MutexFlag) THEN
	RETURN;
END_IF

IF mIsEmpty() THEN
	MutexFlag := FALSE;
	RETURN;
END_IF

IF NOT mCheckHead() THEN
	MutexFlag := FALSE;
	RETURN;
END_IF


mCheck := pBufferPool + HeadIndex * ElementSize;

UsedSize := UsedSize - 1;
IF NOT mIsEmpty() THEN
	HeadIndex := (HeadIndex + 1) MOD NumElements;	
END_IF



MutexFlag := FALSE;
END_METHOD

METHOD PRIVATE mCheckHead : BOOL
VAR_INPUT
END_VAR
VAR
	pDelayedCmdInfo : POINTER TO DelayInfo_typ;
	LogStr : STRING;
END_VAR
VAR_INST
	CmdTimer : StopWatch;
END_VAR

IF mIsEmpty() THEN
	RETURN;
END_IF

pDelayedCmdInfo := (pBufferPool + (HeadIndex * ElementSize));


CASE pDelayedCmdInfo^.DelayType OF
			
	eDelayType.Immediate: 
		mCheckHead := TRUE;
	
	eDelayType.DelayByPos:
		
		IF (Position >= pDelayedCmdInfo^.DelayValue) THEN
			LogStr := CONCAT(Name, 'rid=');
			LogStr := CONCAT(LogStr , UDINT_TO_STRING(pDelayedCmdInfo^.RequestId));
			LogStr := CONCAT(LogStr , ', now=');
			LogStr := CONCAT(LogStr , ULINT_TO_STRING(Position));
			LogStr := CONCAT(LogStr , ', target=');
			LogStr := CONCAT(LogStr , ULINT_TO_STRING(pDelayedCmdInfo^.DelayValue));
			fnLogMsg(ADR(rLogMsg), LOG_INFO, LogStr,0,0,0);
			pDelayedCmdInfo^.LagError := ULINT_TO_UDINT(Position - pDelayedCmdInfo^.DelayValue);
			mCheckHead := TRUE;
		END_IF
		
	eDelayType.DelayByTimer: 
	
		IF NOT CmdTimer.IsActive() THEN
			CmdTimer.Start();
		END_IF
		
		IF TIME_TO_ULINT(CmdTimer.ElapledTime()) >= pDelayedCmdInfo^.DelayValue THEN
			mCheckHead := TRUE;
		END_IF
	
END_CASE

IF mCheckHead THEN
	pDelayedCmdInfo^.Executed := TRUE;
	IF (pDelayedCmdInfo^.pExecuted <> 0) THEN
		pDelayedCmdInfo^.pExecuted^ := TRUE;
	END_IF
	
	IF pDelayedCmdInfo^.DelayType <> eDelayType.DelayByTimer THEN
		CmdTimer.Stop();
	END_IF

END_IF
END_METHOD

METHOD PUBLIC mClear : BOOL
VAR_INPUT
END_VAR
IF NOT TestAndSet(MutexFlag) THEN
	RETURN;
END_IF

TailIndex := HeadIndex := 0;
UsedSize := 0;

mClear := TRUE;

MutexFlag := FALSE;
END_METHOD

METHOD PUBLIC mFront : PVOID // will return true only when next cmd will be ready (time/pos is up)
VAR_INPUT
END_VAR

IF NOT TestAndSet(MutexFlag) THEN
	RETURN;
END_IF

IF mIsEmpty() THEN
	MutexFlag := FALSE;
	RETURN;
END_IF

mFront := pBufferPool + HeadIndex * ElementSize;

MutexFlag := FALSE;
END_METHOD

METHOD PRIVATE mInit : BOOL
VAR_INPUT
END_VAR

mClear();

NumElements := BufferSize/ElementSize;

mInit := TRUE;
END_METHOD

METHOD PUBLIC mIsEmpty : BOOL
VAR_INPUT
END_VAR
mIsEmpty := (UsedSize = 0);
END_METHOD

METHOD PUBLIC mIsFull : BOOL
VAR_INPUT
END_VAR
mIsFull := (UsedSize >= NumElements);
END_METHOD

END_FUNCTION_BLOCK

// ---- POUs/Lib/System/fAnalogSensorScale.TcPOU
FUNCTION fAnalogSensorScale : INT
VAR_INPUT
	IN:INT;
	ptr:POINTER TO AnalogSensorCalibrationTyp;
END_VAR
VAR
	M:REAL;
	B:REAL;
	TEMPX:REAL;
END_VAR

TEMPX := (ptr^.X2-ptr^.X1);
IF TEMPX<>0 THEN
	M:=(ptr^.Y2-ptr^.Y1)/(ptr^.X2-ptr^.X1);
END_IF

IF ptr^.X1 <> 0 AND M <>0 THEN
	B:= ptr^.Y1-(M*ptr^.X1);
	fAnalogSensorScale := REAL_TO_INT(M*IN+B);
ELSIF ptr^.X2 <> 0 AND M <>0 THEN
	B:= ptr^.Y2-(M*ptr^.X1);
	fAnalogSensorScale := REAL_TO_INT(M*IN+B);
END_IF

END_FUNCTION

// ---- POUs/Lib/System/FB_FileEntireReadAtomic.TcPOU

// Read entire fole contents as "atomic" operation encapsulating all required
// file access operations, so no file remain open after the operation completion
// The file data may be read to the buffer provided by calling application or if
// the buffer is not provided or is smaller than file size a dydnamic buffer is
// allocated and its address is returned over outrput parameters and
// it is on duty of the calling application to release the buffer via __DELETE
// when it will not be more needed
// See parameters desctription for more details
FUNCTION_BLOCK FB_FileEntireReadAtomic EXTENDS fb_BaseFb
VAR_INPUT
	sLogThreadName		: STRING := '';	// if not empty, this is thread name to report logs with
	sLogComment			: STRING := '';	// if not empty, is leading each log 
	bExecute	: BOOL;			// operation is started on rising edge of it
	sNetId		: T_AmsNetId := ''; // see FB_FileOpen for details
	sPathName	: T_MaxString;
	ePath		: E_OpenPath := PATH_GENERIC;	 // see FB_FileOpen for details
	tTimeout	: TIME := T#5S;
	
	pRdBufOpt	: POINTER TO BYTE;	// optional Buffer to read data to:
									// if not 0 and rdBufSize >= fileSize, use this bufer to read the data
									// otherwize a new buffer is allocated via _NEW, file is read there
									// and its address is returned in pDataBuf
									// see pDataBuf description for more detals
	rdBufSize	: UDINT := 0;		// see pRdBufOpt for details
END_VAR
VAR_OUTPUT
	bDone				: BOOL;				// becomes TRUE when completed
	bOpError			: BOOL;				// Error encountered and no valid data read
	fileSize			: UDINT;			// returns actual file size / read data size	
	pDataBuf			: POINTER TO BYTE;	// if bOpError is FALSE, this is pointer to the buffer containig entire file data.
											// if bNewRdBufAllocated is FALSE, pDataBuf equals to pRdBufOpt.
											// if bNewRdBufAllocated is TRUE, pDataBuf will point to a buffer
											// allocated via __NEW and newRdBufSize returns this buffer size, which is >= fileSize.
											// It is on duty of application to release the buffer via __DELETE thereafter
											// in order to avoid memory leak											
	bNewRdBufAllocated	: BOOL := FALSE;	// new buffer has been allocated for data and pDataBuf points to it
	newRdBufSize		: UDINT;			// Size of data buffer, which is >= fileSize; See pDataBuf for details 
END_VAR

VAR CONSTANT
	FILE_INACTIVE	: DINT := 0;
	FILE_OPEN		: DINT := 1;
	FILE_SEKK_END	: DINT := 11;
	FILE_SIZE		: DINT := 21;
	FILE_REWIND		: DINT := 31;
	FILE_READ		: DINT := 41;
	FILE_CLOSE		: DINT := 51;
END_VAR

VAR
	executeTrig: Trigger;

	hFile					: UINT := 0;
	FILE_Phase 				: DINT := 0;
	FILE_PhaseAfter_CLOSE	: DINT := 0;
	bOpExec					: BOOL := FALSE;;
END_VAR


IF (executeTrig.EDGEPOS(bExecute)) THEN
	IF (sLogThreadName <>'') THEN
		SetLoggerCategoryName(sLogThreadName);
	END_IF
	IF (sLogComment <>'' AND RIGHT(sLogComment, 1) <> ':') THEN
		CONCAT(sLogComment, ': ');
	END_IF
	bOpError	:= FALSE;
	bDone		:= FALSE;
	IF (hFile = 0) THEN
		FILE_Phase	:= FILE_OPEN;
		bOpExec		:= TRUE;
	ELSE
		LogInfo_v2('%sClose the active fd=%d before opening file %s', hFile, sPathName, DINT_0, DINT_0, DINT_0, DINT_0, DINT_0, DINT_0, DINT_0, DINT_0);
		FILE_Phase				:= FILE_CLOSE;
		FILE_PhaseAfter_CLOSE	:= FILE_OPEN;
		bOpExec					:= (FILE_Phase <> FILE_CLOSE);
	END_IF
END_IF

CASE FILE_Phase OF
	FILE_INACTIVE:
		bDone	:= TRUE;
		
	FILE_OPEN:
		FILE_PhaseAfter_CLOSE	:= FILE_INACTIVE;
		IF (FileOpen()) THEN
			bOpExec		:= TRUE;
			IF (NOT bOpError) THEN
				FILE_Phase	:= FILE_SEKK_END;
			ELSE
				FILE_Phase	:= FILE_INACTIVE;
			END_IF
		END_IF
	FILE_SEKK_END:
		IF (FileSeek(nSeekPos := 0, eOrigin := SEEK_END)) THEN
			bOpExec		:= TRUE;
			IF (NOT bOpError) THEN
				FILE_Phase	:= FILE_SIZE;
			ELSE
				FILE_Phase	:= FILE_CLOSE;
			END_IF
		END_IF
	FILE_SIZE:
		IF (FilePosGet(filePos => fileSize)) THEN
			bOpExec		:= TRUE;
			IF (NOT bOpError) THEN
				FILE_Phase	:= FILE_REWIND;
			ELSE
				FILE_Phase	:= FILE_CLOSE;
			END_IF
		END_IF
	FILE_REWIND:
		IF (FileSeek(nSeekPos := 0, eOrigin := SEEK_SET)) THEN
			bOpExec		:= TRUE;
			// if no error rewinding the file,
			// set/allocate buffer of appropruate size
			IF (NOT bOpError AND_THEN SetDataBuffer()) THEN
				FILE_Phase	:= FILE_READ;
			ELSE
				FILE_Phase	:= FILE_CLOSE;
			END_IF
		END_IF
	FILE_READ:
		IF (FileRead()) THEN
			bOpExec		:= TRUE;
			FILE_Phase	:= FILE_CLOSE;
			IF (bOpError AND bNewRdBufAllocated) THEN
				__DELETE(pDataBuf);
				LogInfo_v2('%sBecause of read error the just allocated buffer was released. File %s', sLogComment, sPathName, DINT_0, DINT_0, DINT_0, DINT_0, DINT_0, DINT_0, DINT_0, DINT_0);
				bNewRdBufAllocated	:= FALSE;
				pDataBuf			:= 0;
				newRdBufSize		:= 0;
			END_IF
		END_IF
	FILE_CLOSE:
		IF (FileClose()) THEN
			bOpExec		:= TRUE;
			FILE_Phase	:= FILE_PhaseAfter_CLOSE;
		END_IF
END_CASE

METHOD PRIVATE FileClose : BOOL
VAR_INST
	fbFileClose	: FB_FileClose;
END_VAR
FileClose := FALSE;

IF (bOpExec) THEN
	fbFileClose(	bExecute	:= FALSE
				, hFile 	:= hFile
				, sNetId	:= sNetId
				, tTimeout	:= T#1S
			);
END_IF

fbFileClose(bExecute := bOpExec);
bOpExec := FALSE;

IF (fbFileClose.bBusy) THEN
	RETURN;
END_IF

FileClose	:= TRUE;
hFile		:= 0;

IF (fbFileClose.bError) THEN
	bOpError := TRUE;
	LogError_v2('%sError 0x%x close fd=%d file %s', sLogComment, fbFileClose.nErrId, fbFileClose.hFile, sPathName
				, DINT_0, DINT_0, DINT_0, DINT_0, DINT_0, DINT_0);
ELSE
	LogInfo_v2('%sDone close fd=%u file %s', sLogComment, fbFileClose.hFile, sPathName
				, DINT_0, DINT_0, DINT_0, DINT_0, DINT_0, DINT_0, DINT_0); 
END_IF
END_METHOD

METHOD PRIVATE FileOpen : BOOL
VAR_INST
	fbFileOpen		: FB_FileOpen;
END_VAR
fileOpen := FALSE;

IF (bOpExec) THEN
	fbFileOpen(	bExecute	:= FALSE
				, ePath		:= ePath
				, nMode		:= FOPEN_MODEREAD OR FOPEN_MODEBINARY
				, sPathName	:= sPathName
				, sNetId	:= sNetId
				, tTimeout	:=  tTimeout
			);
END_IF

fbFileOpen(bExecute := bOpExec);
bOpExec := FALSE;

IF (fbFileOpen.bBusy) THEN
	RETURN;
END_IF

fileOpen := TRUE;

IF (fbFileOpen.bError) THEN
	bOpError := TRUE;
	LogError_v2('%sError 0x%x open file %s', sLogComment, fbFileOpen.nErrId, fbFileOpen.sPathName
				, DINT_0, DINT_0, DINT_0, DINT_0, DINT_0, DINT_0, DINT_0); 
ELSE
	hFile := fbFileOpen.hFile;
	LogInfo_v2('%sDone open fd=%d file %s', sLogComment, fbFileOpen.hFile, fbFileOpen.sPathName
				, DINT_0, DINT_0, DINT_0, DINT_0, DINT_0, DINT_0, DINT_0); 
END_IF
END_METHOD

METHOD PRIVATE FilePosGet : BOOL
VAR_OUTPUT
	filePos		: UDINT;
END_VAR
VAR_INST
	fbFileTell	: FB_FileTell;
END_VAR
FilePosGet := FALSE;

IF (bOpExec) THEN
	fbFileTell(	bExecute	:= FALSE
				, hFile 	:= hFile
				, sNetId	:= sNetId
				, tTimeout	:=  T#1S
			);
END_IF

fbFileTell(bExecute := bOpExec);
bOpExec := FALSE;

IF (fbFileTell.bBusy) THEN
	RETURN;
END_IF

FilePosGet := TRUE;

IF (fbFileTell.bError) THEN
	bOpError := TRUE;
	LogError_v2('%sError 0x%x get pos of file %s', sLogComment, fbFileTell.nErrId, sPathName
				, DINT_0, DINT_0, DINT_0, DINT_0, DINT_0, DINT_0, DINT_0);
ELSE
	 filePos	:= DINT_TO_UDINT(fbFileTell.nSeekPos);
END_IF
END_METHOD

METHOD PRIVATE FileRead : BOOL
VAR_INST
	fbFileRead	: FB_FileRead;
END_VAR
FileRead := FALSE;

IF (bOpExec) THEN
	fbFileRead(	bExecute	:= FALSE
				, hFile 	:= hFile
				, pReadBuff	:= pDataBuf                        
				, cbReadLen	:= FileSize                    
				, sNetId	:= sNetId
				, tTimeout	:= tTimeout
			);
END_IF

fbFileRead(bExecute := bOpExec);
bOpExec := FALSE;

IF (fbFileRead.bBusy) THEN
	RETURN;
END_IF

FileRead := TRUE;

IF (fbFileRead.bError OR fbFileRead.cbRead <> fbFileRead.cbReadLen) THEN
	bOpError := TRUE;
	LogError_v2('%sError 0x%x read rqst=%u act=%u bytes from file %s', sLogComment, fbFileRead.nErrId, fbFileRead.cbReadLen, fbFileRead.cbRead, sPathName
				, DINT_0, DINT_0, DINT_0, DINT_0, DINT_0);
ELSE
	LogInfo_v2('%sDone read %u bytes from file %s', sLogComment, fbFileRead.cbRead, sPathName
				, DINT_0, DINT_0, DINT_0, DINT_0, DINT_0, DINT_0, DINT_0); 
END_IF
END_METHOD

METHOD PRIVATE FileSeek : BOOL
VAR_INPUT
	nSeekPos	: DINT;
	eOrigin		: E_SeekOrigin:= SEEK_SET;
END_VAR
VAR_INST
	fbFileSeek	: FB_FileSeek;
END_VAR
FileSeek := FALSE;

IF (bOpExec) THEN
	fbFileSeek(	bExecute	:= FALSE
				, hFile 	:= hFile
				, eOrigin	:= eOrigin
				, nSeekPos	:= nSeekPos
				, sNetId	:= sNetId
				, tTimeout	:=  T#1S
			);
END_IF

fbFileSeek(bExecute := bOpExec);
bOpExec := FALSE;

IF (fbFileSeek.bBusy) THEN
	RETURN;
END_IF

FileSeek := TRUE;

IF (fbFileSeek.bError) THEN
	bOpError := TRUE;
	LogError_v2('%sError 0x%x seek pos=%u origin=%u file %s', sLogComment, fbFileSeek.nErrId, fbFileSeek.nSeekPos, fbFileSeek.eOrigin, sPathName
				, DINT_0, DINT_0, DINT_0, DINT_0, DINT_0); 
END_IF
END_METHOD

METHOD PRIVATE SetDataBuffer : BOOL
VAR
	bufSizeRound	: UDINT := 16#100000;
END_VAR

SetDataBuffer	:= TRUE;

bNewRdBufAllocated	:= FALSE;
pDataBuf			:= pRdBufOpt;
newRdBufSize		:= 0;

IF (pDataBuf <> 0 AND rdBufSize >= fileSize) THEN
	RETURN;
END_IF

LogInfo_v2('%sAlloc buf to read the file (fSize=%u), since user buf is short (size=%u) or not set:  file %s', sLogComment, fileSize, rdBufSize, sPathName
			, DINT_0, DINT_0, DINT_0, DINT_0, DINT_0, DINT_0);
			
// allocate buffer to read the file
newRdBufSize	:= (((fileSize+1) + (bufSizeRound-1)) / bufSizeRound) * bufSizeRound;
pDataBuf		:= __NEW (BYTE, newRdBufSize);
IF (pDataBuf = 0) THEN
	SetDataBuffer	:= FALSE;
	bOpError		:= TRUE;
	LogError_v2('%sError: mem alloc size=%u to read file %s', sLogComment, newRdBufSize, sPathName
				, DINT_0, DINT_0, DINT_0, DINT_0, DINT_0, DINT_0, DINT_0);
	newRdBufSize	:= 0;
ELSE
	bNewRdBufAllocated	:= TRUE;
	LogInfo_v2('%sDone buf alloc size=%u to read file %s', sLogComment, newRdBufSize, sPathName
				, DINT_0, DINT_0, DINT_0, DINT_0, DINT_0, DINT_0, DINT_0);
END_IF
END_METHOD

END_FUNCTION_BLOCK

// ---- GlobalTextList.TcGTLO
TEXTLIST GlobalTextList
  546 = '%5.2f'
  22 = '%s'
  525 = 'Advance'
  35 = 'Back'
  942 = 'Close Valves'
  956 = 'Cold Cut'
  835 = 'Cold Cut Piston'
  646 = 'Cold Cut Valve'
  321 = 'Continues'
  837 = 'Continunes'
  509 = 'Corona'
  359 = 'Cycles Number %d'
  221 = 'Dancer Full '
  339 = 'Diameter %5.0f'
  966 = 'Diameter %5.2f'
  386 = 'Diameter %d'
  485 = 'E-Stop'
  561 = 'E-Stop Pressed'
  918 = 'Empty'
  479 = 'Enable Dancer'
  425 = 'End Position'
  553 = 'EndPosition'
  650 = 'External Nip'
  119 = 'Forward'
  185 = 'Full'
  511 = 'Gripper Close'
  235 = 'Gripper Open'
  855 = 'Gripper Open/Close'
  294 = 'Gripper Position'
  447 = 'Gripper Retract'
  809 = 'Gripper Retract/Extract'
  721 = 'Grpper Position'
  828 = 'Heater Off'
  824 = 'Heater On'
  562 = 'Heater On '
  744 = 'Home'
  757 = 'Hot Welding'
  134 = 'Hot Welding Off'
  18 = 'Hot Welding On'
  373 = 'Hot Welding On/Off'
  560 = 'IO'
  96 = 'IO_1'
  128 = 'Jog +'
  619 = 'Jog -'
  573 = 'Jog Both  -'
  332 = 'Jog Both +'
  508 = 'Knive Cut'
  714 = 'Limit'
  911 = 'machine state'
  649 = 'Machine State'
  979 = 'Machine State %s'
  219 = 'Machine State %S'
  23 = 'Machine State - %s'
  759 = 'Manual'
  363 = 'Motor On'
  27 = 'None'
  549 = 'OFF'
  698 = 'OK'
  246 = 'Output'
  476 = 'Output gripper'
  667 = 'Press Down'
  387 = 'Press Down Time'
  227 = 'Press Up/Down'
  488 = 'Press UpTime'
  8 = 'Press Valve'
  980 = 'Restart'
  605 = 'Session Counter'
  143 = 'Session Counter - %d'
  925 = 'Set Time [MS] %d'
  851 = 'Simulation'
  1 = 'Speed'
  800 = 'Start'
  772 = 'Start Position'
  483 = 'Stop'
  801 = 'Tension %5.0f'
  566 = 'Timer Set Time %d'
  290 = 'Timer Set Time [ms] %d'
  702 = 'UW 1'
  633 = 'UW 2'
  83 = 'Valves Close'
  155 = 'Welding Piston'
  640 = 'Welding Valve'
  439 = 'Winders'
END_TEXTLIST

// ---- VISUs/Dialogs/DialogTimer.TcVIS
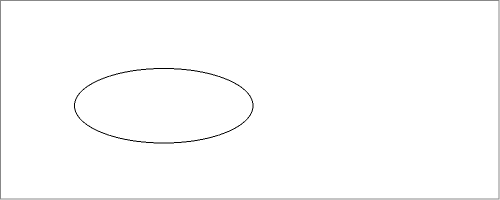
VISUALIZATION DialogTimer  // 500x200
    Ellipse (74,68 179x75)
END_VISUALIZATION

// ---- VISUs/Dialogs/DialogTimer_ColdCut.TcVIS
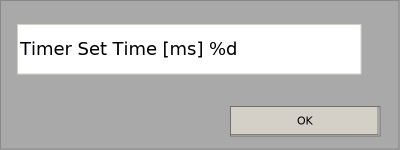
VISUALIZATION DialogTimer_ColdCut  // 400x150
    Button (230,106 150x30), "OK"
        OnMouseClick: CloseDialog Dialog=DialogTimer_ColdCut, Result=OK, NumpadKeypadSet=True
    Textfield (17,24 344x50), "Timer Set Time [ms] %d", text variable: PersistentStruct.TimeColdCutPressDown
        OnMouseClick: write the text variable via Edit
END_VISUALIZATION

// ---- VISUs/Dialogs/DialogTimer_GripperPosi.TcVIS
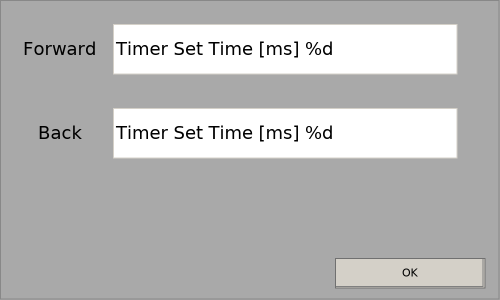
VISUALIZATION DialogTimer_GripperPosi  // 500x300
    Button (335,258 150x30), "OK"
        OnMouseClick: CloseDialog Dialog=DialogTimer_GripperPosi, Result=OK, NumpadKeypadSet=True
    Textfield (113,24 344x50), "Timer Set Time [ms] %d", text variable: PersistentStruct.TimeGripperStartPosition
        OnMouseClick: write the text variable via Edit
    Textfield (113,108 344x50), "Timer Set Time [ms] %d", text variable: PersistentStruct.TimeGripperHomePosition
        OnMouseClick: write the text variable via Edit
    Label (4,34 112x30), "Forward"
    Label (4,118 112x30), "Back"
END_VISUALIZATION

// ---- VISUs/Dialogs/DialogTimer_HeaterOff.TcVIS
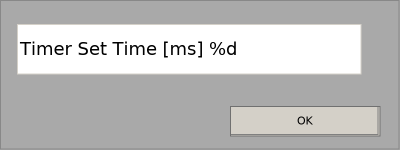
VISUALIZATION DialogTimer_HeaterOff  // 400x150
    Button (230,106 150x30), "OK"
        OnMouseClick: CloseDialog Dialog=DialogTimer_HeaterOff, Result=OK, NumpadKeypadSet=True
    Textfield (17,24 344x50), "Timer Set Time [ms] %d", text variable: PersistentStruct.TimerHotWeldingOff
        OnMouseClick: write the text variable via Edit
END_VISUALIZATION

// ---- VISUs/Dialogs/DialogTimer_GripperOpenClose.TcVIS
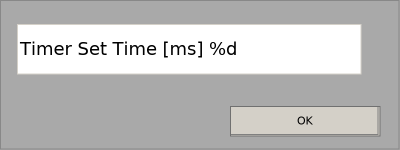
VISUALIZATION DialogTimer_GripperOpenClose  // 400x150
    Button (230,106 150x30), "OK"
        OnMouseClick: CloseDialog Dialog=DialogTimer_GripperOpenClose, Result=OK, NumpadKeypadSet=True
    Textfield (17,24 344x50), "Timer Set Time [ms] %d", text variable: PersistentStruct.TimeGripperOpen
        OnMouseClick: write the text variable via Edit
END_VISUALIZATION

// ---- VISUs/Dialogs/DialogTimer_HotWeldValve.TcVIS
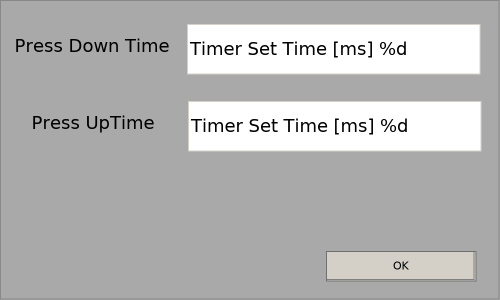
VISUALIZATION DialogTimer_HotWeldValve  // 500x300
    Button (326,251 150x30), "OK"
        OnMouseClick: CloseDialog Dialog=DialogTimer_HotWeldValve, Result=OK, NumpadKeypadSet=True
    Textfield (187,24 293x50), "Timer Set Time [ms] %d", text variable: PersistentStruct.TimeHotWeldPressDown
        OnMouseClick: write the text variable via Edit
    Label (6,31 172x30), "Press Down Time"
    Textfield (188,101 293x50), "Timer Set Time [ms] %d", text variable: PersistentStruct.TimerPressUp
        OnMouseClick: write the text variable via Edit
    Label (7,108 172x30), "Press UpTime"
END_VISUALIZATION

// ---- VISUs/Dialogs/DialogTimer_HeaterOn.TcVIS
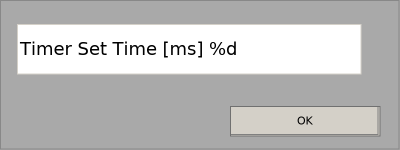
VISUALIZATION DialogTimer_HeaterOn  // 400x150
    Button (230,106 150x30), "OK"
        OnMouseClick: CloseDialog Dialog=DialogTimer_HeaterOn, Result=OK, NumpadKeypadSet=True
    Textfield (17,24 344x50), "Timer Set Time [ms] %d", text variable: PersistentStruct.TimerHotWeldingOn
        OnMouseClick: write the text variable via Edit
END_VISUALIZATION

// ---- VISUs/Dialogs/DialogTimer_ValveClose.TcVIS
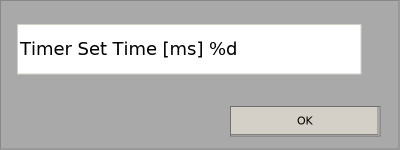
VISUALIZATION DialogTimer_ValveClose  // 400x150
    Button (230,106 150x30), "OK"
        OnMouseClick: CloseDialog Dialog=DialogTimer_ValveClose, Result=OK, NumpadKeypadSet=True
    Textfield (17,24 344x50), "Timer Set Time [ms] %d", text variable: PersistentStruct.TimeGripperRetract
        OnMouseClick: write the text variable via Edit
END_VISUALIZATION

// ---- VISUs/Dialogs/Dialog_Estop.TcVIS
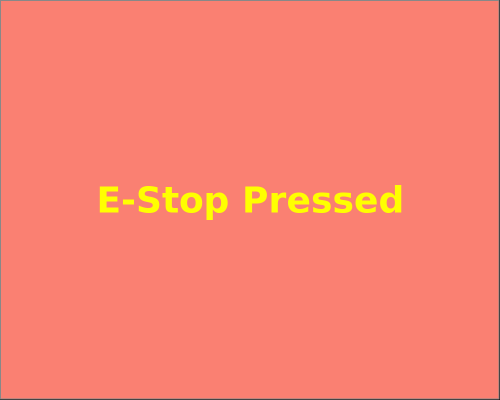
VISUALIZATION Dialog_Estop  // 500x400
    Rectangle (0,0 500x400), colour toggle: HMI.EstopDialogBackgroundColor
    Label (99,137 303x126), "E-Stop Pressed"
END_VISUALIZATION

// ---- VISUs/Dialogs/Dialog_IO.TcVIS
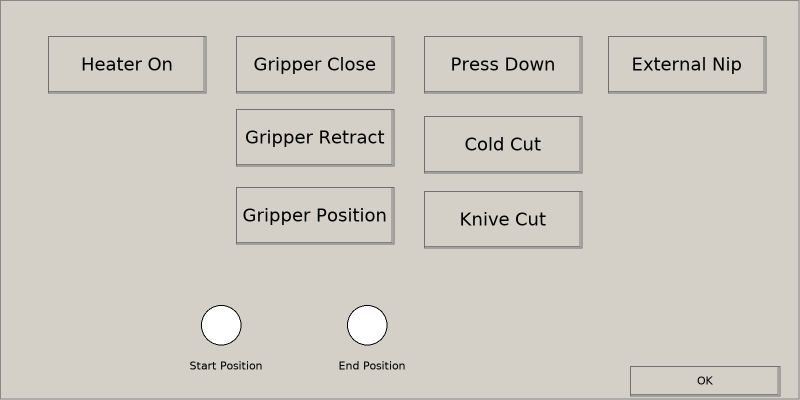
VISUALIZATION Dialog_IO  // 800x400
    Button (48,36 158x57), "Heater On"
        toggle gMachineCtrl.IO.Out.HeaterOn
    Button (236,36 158x57), "Gripper Close"
        toggle gMachineCtrl.IO.Out.GripperOpen
    Button (236,109 158x57), "Gripper Retract"
        toggle gMachineCtrl.IO.Out.GripperRetract
    Button (236,187 158x57), "Gripper Position"
        toggle gMachineCtrl.IO.Out.GripperPistonPosition
    Button (424,36 158x57), "Press Down"
        toggle gMachineCtrl.IO.Out.PressDown
    Button (630,366 150x30), "OK"
        OnMouseDown: CloseDialog Dialog=Dialog_IO, Result=OK, NumpadKeypadSet=True
    Button (608,36 158x57), "External Nip"
        toggle gMachineCtrl.IO.Out.ExternalNipMotor
    Ellipse (201,305 40x40), colour toggle: gMachineCtrl.IO.In.GripperStartPosition
    Label (171,351 110x30), "Start Position"
    Ellipse (347,305 40x40), colour toggle: gMachineCtrl.IO.In.GripperStartPosition
    Label (317,351 110x30), "End Position"
    Button (424,116 158x57), "Cold Cut"
        toggle gMachineCtrl.IO.Out.ColdCutPistonDown
    Button (424,191 158x57), "Knive Cut"
        toggle gMachineCtrl.IO.Out.KniveCut
END_VISUALIZATION

// ---- VISUs/Dialogs/Dialog_Output.TcVIS
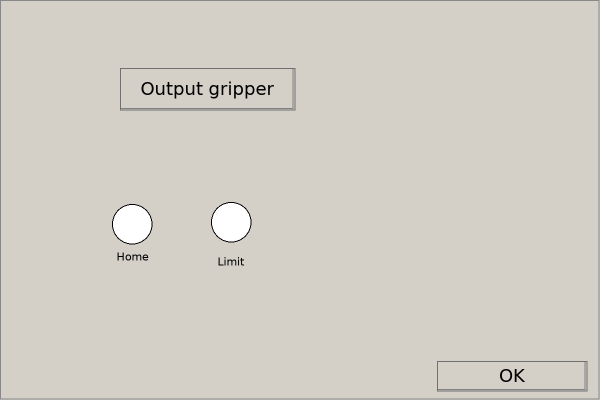
VISUALIZATION Dialog_Output  // 600x400
    Button (437,361 150x30), "OK"
        OnMouseClick: CloseDialog Dialog=Dialog_Output, Result=OK, NumpadKeypadSet=True
    Ellipse (112,204 40x40), colour toggle: gMachineCtrl.IO.In.HomeOutAxis
    Button (120,68 175x42), "Output gripper"
        toggle gMachineCtrl.IO.Out.Output_GripperClose
    Ellipse (211,202 40x40), colour toggle: gMachineCtrl.IO.In.HomeOutAxisLimit
    Label (102,242 62x30), "Home"
    Label (200,247 62x30), "Limit"
END_VISUALIZATION

// ---- VISUs/Dialogs/Dialog_Settings.TcVIS
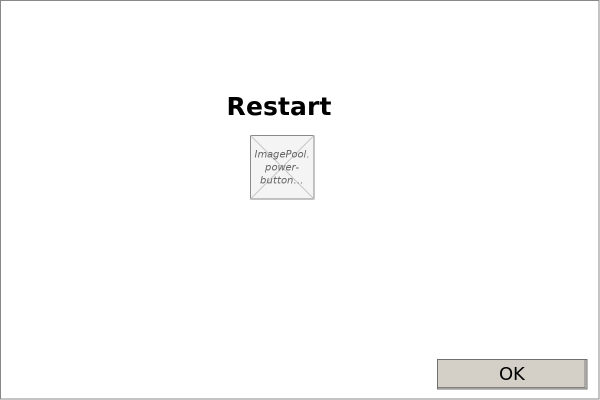
VISUALIZATION Dialog_Settings  // 600x400
    Button (437,359 150x30), "OK"
        OnMouseClick: CloseDialog Dialog=Dialog_Settings, Result=OK, NumpadKeypadSet=True
    Image (250,135 64x64), image: ImagePool.power-button-svgrepo-com
        OnMouseClick: toggle HMI.TC_Restart.RESTART
    Label (204,91 150x30), "Restart"
END_VISUALIZATION

// ---- VISUs/Dialogs/Winders.TcVIS
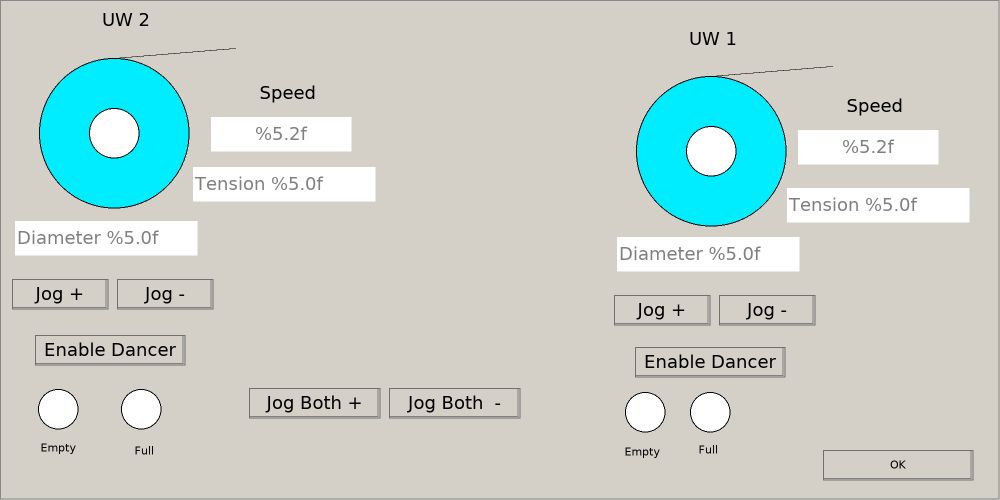
VISUALIZATION Winders  // 1000x500
    Button (823,450 150x30), "OK"
        OnMouseDown: CloseDialog Dialog=Winders, Result=OK, NumpadKeypadSet=True
    Ellipse (636,76 150x150)
    Ellipse (686,126 50x50)
    Line (698,77) (832,66)
    Ellipse (39,58 150x150)
    Ellipse (89,108 50x50)
    Line (101,59) (235,48)
    Label (638,24 150x30), "UW 1"
    Label (51,5 150x30), "UW 2"
    Textfield (616,236 184x36), "Diameter %5.0f", text variable: prg_Motion.UW_1_Diameter.Diameter_filtred
        OnMouseClick: write the text variable via Edit, min 0, max 1000000, title "Enter number of cycles"
    Button (614,295 96x30), "Jog +"
        tap gMachineCtrl.Cmd.UW_1_Cmd.JogSFwdSlow
    Button (719,295 96x30), "Jog -"
        tap gMachineCtrl.Cmd.UW_1_Cmd.JogBackdSlow
    Textfield (797,129 142x36), "%5.2f", text variable: gWebAxes.UW_1.Ref.NcToPlc.ActVelo
        OnMouseClick: write the text variable via Edit, min 0, max 1000000, title "Enter number of cycles"
    Label (800,91 150x30), "Speed"
    Textfield (210,116 142x36), "%5.2f", text variable: gWebAxes.UW_2.Ref.NcToPlc.ActVelo
        OnMouseClick: write the text variable via Edit, min 0, max 1000000, title "Enter number of cycles"
    Label (213,78 150x30), "Speed"
    Textfield (14,220 184x36), "Diameter %5.0f", text variable: prg_Motion.UW_2_Diameter.Diameter_filtred
        OnMouseClick: write the text variable via Edit, min 0, max 1000000, title "Enter number of cycles"
    Button (12,279 96x30), "Jog +"
        tap gMachineCtrl.Cmd.UW_2_Cmd.JogSFwdSlow
    Button (117,279 96x30), "Jog -"
        tap gMachineCtrl.Cmd.UW_2_Cmd.JogBackdSlow
    Button (249,388 131x30), "Jog Both +"
        OnMouseDown: execute { gMachineCtrl.Cmd.UW_2_Cmd.JogSFwdSlow := TRUE; gMachineCtrl.Cmd.UW_1_Cmd.JogSFwdSlow := TRUE; }
        OnMouseUp: execute { gMachineCtrl.Cmd.UW_2_Cmd.JogSFwdSlow := FALSE; gMachineCtrl.Cmd.UW_1_Cmd.JogSFwdSlow := FALSE; }
    Button (389,388 131x30), "Jog Both -"
        OnMouseDown: execute { gMachineCtrl.Cmd.UW_2_Cmd.JogBackdSlow := TRUE; gMachineCtrl.Cmd.UW_1_Cmd.JogBackdSlow := TRUE; }
        OnMouseUp: execute { gMachineCtrl.Cmd.UW_2_Cmd.JogBackdSlow := FALSE; gMachineCtrl.Cmd.UW_1_Cmd.JogBackdSlow := FALSE; }
    Textfield (786,187 184x36), "Tension %5.0f", text variable: prg_Motion.UW_1_Data.Tension.Tension_filtred
    Textfield (192,166 184x36), "Tension %5.0f", text variable: prg_Motion.UW_2_Data.Tension.Tension_filtred
    Button (35,335 150x30), "Enable Dancer"
        toggle gMachineCtrl.Parameters.UW_2_Param.EnableDancer
    Button (635,347 150x30), "Enable Dancer"
        toggle gMachineCtrl.Parameters.UW_1_Param.EnableDancer
    Ellipse (121,389 40x40), colour toggle: gMachineCtrl.IO.In.UW_2_DancerFull
    Ellipse (690,392 40x40), colour toggle: gMachineCtrl.IO.In.UW_1_DancerFull
    Ellipse (38,389 40x40), colour toggle: gMachineCtrl.IO.In.UW_2_DancerEmpety
    Label (27,433 63x30), "Empty"
    Label (113,436 63x30), "Full"
    Ellipse (625,392 40x40), colour toggle: gMachineCtrl.IO.In.UW_1_DancerEmpety
    Label (677,435 63x30), "Full"
    Label (611,437 63x30), "Empty"
END_VISUALIZATION

// ---- VISUs/Img/MachineState.TcTLO
TEXTLIST MachineState
  10 = 'Off'
  20 = 'Run'
  0 = 'Init'
   = ''
END_TEXTLIST

// ---- VISUs/Visualization.TcVIS
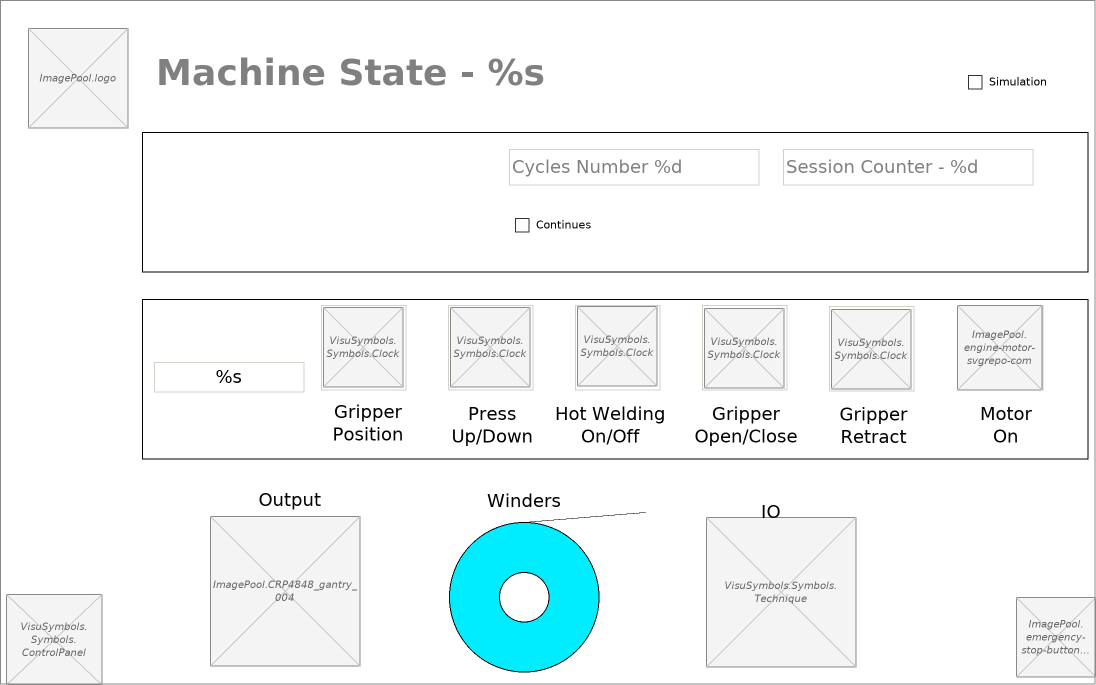
VISUALIZATION Visualization  // 1096x685
    RoundedRectangle (142,299 946x160)
    RoundedRectangle (142,132 946x140)
    Image (28,28 100x100), image: ImagePool.logo
        p2858320360: HMI.LogoRotation
    RoundedRectangle (267,147 100x100), colour toggle: HMI.StartButtonColor
    Image (278,159 75x75), image: ImagePool.play-button-svgrepo-com
    RoundedRectangle (268,147 100x100)
        tap gMachineCtrl.Cmd.Start
        OnMouseEnter: toggle HMI.StartButtonColor
        OnMouseLeave: toggle HMI.StartButtonColor
    Group (378,147 100x100)
        RoundedRectangle (0,0 100x100), colour toggle: HMI.StopButtonColor
        Image (14,12 75x75), image: ImagePool.stop-svgrepo-com
        RoundedRectangle (0,0 100x100)
            tap gMachineCtrl.Cmd.Stop
            OnMouseEnter: toggle HMI.StopButtonColor
            OnMouseLeave: toggle HMI.StopButtonColor
    Textfield (153,41 743x63), "Machine State - %s", text variable: FB_Machine_Ctrl.Monitoring.StepMessage
    Checkbox (513,205 150x40), "Continues", variable: gMachineCtrl.Parameters.Continues
    Textfield (509,149 250x36), "Cycles Number %d", text variable: gMachineCtrl.Parameters.NumberOfCycles, input disabled if: gMachineCtrl.Parameters.Continues
        OnMouseClick: write the text variable via Edit, min 0, max 1000000, title "Enter number of cycles"
    Textfield (783,149 250x36), "Session Counter - %d", text variable: gMachineCtrl.Status.SessionCounter
    Textfield (154,362 150x30), "%s", text variable: FB_Machine_Run.Delay.ET
    RoundedRectangle (321,305 85x85), colour toggle: HMI.TimerGripperPostionColor
    Image (323,307 80x80), image: VisuSymbols.Symbols.Clock
        OnMouseClick: OpenDialog Dialog=DialogTimer_GripperPosi, OpenModal=True, OpenCentered=True
    Label (313,389 110x68), "Gripper Position"
    Label (549,393 123x64), "Hot Welding On/Off"
    Label (685,395 122x60), "Gripper Open/Close"
    Label (824,397 99x57), "Gripper Retract"
    Label (443,386 99x78), "Press Up/Down"
    RoundedRectangle (448,305 85x85), colour toggle: HMI.TimerHotWeldColor
    Image (450,307 80x80), image: VisuSymbols.Symbols.Clock
        OnMouseClick: OpenDialog Dialog=DialogTimer_HotWeldValve, OpenModal=True, OpenCentered=True
    RoundedRectangle (575,305 85x85), colour toggle: HMI.TimerHeaterOnColor
    Image (577,306 80x80), image: VisuSymbols.Symbols.Clock
        OnMouseClick: OpenDialog Dialog=DialogTimer_HeaterOn, OpenModal=True, OpenCentered=True
    RoundedRectangle (702,305 85x85), colour toggle: HMI.TimerGripperopenColor
    Image (704,308 80x80), image: VisuSymbols.Symbols.Clock
        OnMouseClick: OpenDialog Dialog=DialogTimer_GripperOpenClose, OpenModal=True, OpenCentered=True
    RoundedRectangle (829,306 85x85), colour toggle: HMI.TimerGripperRetractColor
    Image (831,309 80x80), image: VisuSymbols.Symbols.Clock
        OnMouseClick: OpenDialog Dialog=DialogTimer_ValveClose, OpenModal=True, OpenCentered=True
    RoundedRectangle (958,305 85x85), colour toggle: HMI.StateMotorOnColor
    Label (972,391 68x68), "Motor On"
    Image (957,305 85x85), image: ImagePool.engine-motor-svgrepo-com
    Image (1016,597 80x80), image: ImagePool.emergency-stop-button-icon-364856
        p1097714728: HMI.EstopScalling
        OnMouseClick: toggle gMachineCtrl.Cmd.EmStop
        OnMouseDown: execute { HMI.EstopScalling	:= 1100; }
        OnMouseUp: execute { HMI.EstopScalling	:= 1300; }
        OnMouseEnter: execute { HMI.EstopScalling	:= 1300; }
        OnMouseLeave: execute { HMI.EstopScalling	:= 1000; }
    Checkbox (966,67 109x30), "Simulation", variable: gMachineCtrl.Simulation
    RoundedRectangle (166,151 100x100), colour toggle: HMI.SwitchOnButtonColor
    Image (185,163 64x64), image: ImagePool.power-power-button-svgrepo-com
        p1097714728: HMI.onOffScaling
    RoundedRectangle (165,150 100x100)
        toggle gMachineCtrl.Cmd.SwitchOn
        OnMouseEnter: execute { HMI.SwitchOnButtonColor :=TRUE; HMI.onOffScaling		:=1200; }
        OnMouseLeave: execute {
            IF gMachineCtrl.Cmd.SwitchOn THEN
            	HMI.SwitchOnButtonColor:=TRUE;
            ELSE
            	HMI.SwitchOnButtonColor:=FALSE;
            END_IF
            HMI.onOffScaling		:=1000;
        }
    Group (449,486 196x186)
        p1097714728: HMI.WinderScaling
        OnMouseClick: OpenDialog Dialog=Winders, OpenModal=True, OpenCentered=True
        OnDialogClosed: execute { HMI.WinderScaling := 1000; }
        OnMouseDown: execute { HMI.WinderScaling := 1000; }
        OnMouseEnter: execute { HMI.WinderScaling := 1100; }
        OnMouseLeave: execute { HMI.WinderScaling := 1000; }
        Label (0,0 150x30), "Winders"
        Ellipse (0,36 150x150)
            OnMouseDown: OpenDialog Dialog=Winders, OpenModal=True, OpenCentered=True
        Ellipse (50,86 50x50)
        Line (62,37) (196,26)
    Image (6,594 96x91), image: VisuSymbols.Symbols.ControlPanel
        p1097714728: HMI.SettingsScaling
        OnMouseClick: OpenDialog Dialog=Dialog_Settings, OpenModal=True, OpenCentered=True
        OnDialogClosed: execute { HMI.SettingsScaling:=1000; }
        OnMouseDown: execute { HMI.SettingsScaling:=1000; }
        OnMouseEnter: execute { HMI.SettingsScaling:=1100; }
        OnMouseLeave: execute { HMI.SettingsScaling:=1000; }
    Group (696,497 160x170)
        p1097714728: HMI.IOScaling
        OnMouseClick: OpenDialog Dialog=Dialog_IO, OpenModal=True, OpenCentered=True
        OnMouseLeave: execute { HMI.IOScaling:=1000; }
        OnDialogClosed: execute { HMI.IOScaling:=1000; }
        OnMouseEnter: execute { HMI.IOScaling:=1150; }
        Image (10,20 150x150), image: VisuSymbols.Symbols.Technique
            OnMouseClick: OpenDialog Dialog=Dialog_IO, OpenModal=True, OpenCentered=True
        Label (0,0 150x30), "IO"
    Label (215,485 150x30), "Output"
    Image (210,516 150x150), image: ImagePool.CRP4848_gantry_004
        OnMouseDown: execute { HMI.OutputScaling:=1000; }
        OnMouseLeave: execute { HMI.OutputScaling:=1000; }
        OnMouseClick: OpenDialog Dialog=Dialog_Output, OpenModal=True, OpenCentered=True
        OnMouseEnter: execute { HMI.OutputScaling:=1100; }
        OnDialogClosed: execute { HMI.OutputScaling:=1000; }
END_VISUALIZATION
